FUNCTION_BLOCK "HOPPER"	// FB 1001
TITLE = HOPPER
//Creation:
//Date:            Author:                                               Version
//--------------------------------------------------------------------------------
//17.04.17          Ilia Bedniakov (ilia   )                             01.00.00
//
//Changes:
//No. Date:        Who       Description                           Mark   Version 
//--------------------------------------------------------------------------------
//01
//________________________________________________________________________________
//Function:
AUTHOR : ilia
VERSION : 0.1
VAR_INPUT
  in_HopperNumber : INT ;
  IF_FC_RotaryFeeder_DB : INT ;	//IF DB number
  IF_FC_RotaryFeeder_DW : INT ;	//start DW of IF structure
  SystemActive : BOOL ;	//system control on
  iLowLevelHopper : BOOL ;
  iRepRotaryFeeder : BOOL ;	//repair switch
  iRepVibrator1 : BOOL ;
  iRepVibrator2 : BOOL ;
  iFBVibrator1_on : BOOL ;
  iFBVibrator2_on : BOOL ;
  iFBRotaryFeeder_on : BOOL ;	//feedback
  iProductValve_open : BOOL ;	//feedback
  iSafetyRotaryFeeder_ok : BOOL ;	//safety switch
  iSafetyToolKeyControl : BOOL ;	//Tool control safety switch
  aFBRotaryFeeder : BOOL ;	//ack feedback fault
  aFBVibrator1 : BOOL ;
  aFBVibrator2 : BOOL ;
  aRepRotaryValve : BOOL ;	//ack repair switch
  aRepVibrator1 : BOOL ;
  aRepVibrator2 : BOOL ;
  aSafetyRotaryFeeder : BOOL ;	//ack safety switch
  aToolKeyControl : BOOL ;	//ack Tool Control
END_VAR
VAR_IN_OUT
  qRotaryFeeder_on : BOOL ;	//output
  qAPBRotaryFeeder : BOOL ;	//output
  qVibrator1 : BOOL ;
  qVibrator2 : BOOL ;
  fFBRotaryFeeder : BOOL ;	//feedback fault
  fFBVibrator1 : BOOL ;
  fFBVibrator2 : BOOL ;
  fRepRotaryFeeder : BOOL ;	//repair switch fault
  fRepVibrator1 : BOOL ;
  fRepVibrator2 : BOOL ;
  fSafetyRotaryFeeder : BOOL ;	//safety fault
  fToolKeyControl : BOOL ;	//rotary control fault
  fProductFlap : BOOL ;
END_VAR
VAR
  reserve_IO : ARRAY  [12 .. 49 ] OF BYTE ;
  HMI : STRUCT 	//Interface of HMI
   CMD : STRUCT
    reserve : BOOL ;
    Vibrator1_man_release : BOOL ;
    Vibrator2_man_release : BOOL ;
    reserve_3 : BOOL ;
    reserve_4 : BOOL ;
    reserve_5 : BOOL ;
    reserve_6 : BOOL ;
    reserve_7 : BOOL ;
    reserve_8 : BOOL ;
    reserve_9 : BOOL ;
    reserve_10 : BOOL ;
    reserve_11 : BOOL ;
    reserve_12 : BOOL ;
    reserve_13 : BOOL ;
    reserve_14 : BOOL ;
    reserve_15 : BOOL ;
   END_STRUCT ;
   STATE : STRUCT
    Active_Discharge : BOOL ;
    reserve_14 : BOOL ;
    reserve_12 : BOOL ;
    DischargingReleased : BOOL ;
    reserve : BOOL ;
    reserve_1 : BOOL ;
    reserve_2 : BOOL ;
    reserve_3 : BOOL ;
    reserve_4 : BOOL ;
    reserve_5 : BOOL ;
    reserve_6 : BOOL ;
    reserve_7 : BOOL ;
    reserve_8 : BOOL ;
    reserve_9 : BOOL ;
    reserve_10 : BOOL ;
    reserve_11 : BOOL ;
   END_STRUCT ;
   PARAM : STRUCT
    SetFrequency : REAL  := 3.000000e+001;
    DelayOn_RotaryValve : REAL  := 3.000000e+000;
    RestDischarge_Time : REAL  := 1.000000e+001;
    reserve_2 : REAL ;
    reserve_3 : INT ;
    reserve_4 : INT ;
    reserve_5 : INT ;
    reserve_6 : INT ;
    reserve_7 : INT ;
    reserve_8 : INT ;
    reserve_9 : REAL  := 1.200000e+002;
    reserve_10 : REAL  := 3.000000e+002;
    reserve_11 : REAL  := 5.000000e+000;
    reserve_12 : REAL  := 1.000000e+001;	//Minutes
    reserve_13 : REAL  := 1.000000e+001;
   END_STRUCT ;
   PV : STRUCT
    actFrequency : REAL ;
    DelayOn_RotaryValve : REAL ;
    RestDischarge_Time : REAL ;
    reserve : REAL ;
    reserve_1 : REAL ;
    reserve_2 : INT ;
    reserve_3 : INT ;
    reserve_4 : INT ;
    reserve_5 : INT ;
    reserve_6 : INT ;
    reserve_7 : INT ;
    reserve_8 : REAL ;
    reserve_9 : REAL ;
    reserve_10 : REAL ;
    reserve_11 : REAL ;	//Minutes
   END_STRUCT ;
  END_STRUCT ;
  PROD : STRUCT 	//Interface of Production
   FROM : STRUCT
    reserve : INT ;
    reserve_1 : INT ;
    reserve_2 : INT ;
    reserve_3 : INT ;
    reserve_4 : INT ;
    reserve_5 : REAL ;
    reserve_6 : REAL ;
    CMD : STRUCT
     reserve : BOOL ;
     reserve_1 : BOOL ;
     reserve_2 : BOOL ;
     reserve_3 : BOOL ;
     reserve_4 : BOOL ;
     reserve_5 : BOOL ;
     reserve_6 : BOOL ;
     reserve_7 : BOOL ;
     reserve_8 : BOOL ;
     reserve_9 : BOOL ;
     reserve_10 : BOOL ;
     reserve_11 : BOOL ;
     reserve_12 : BOOL ;
     reserve_13 : BOOL ;
     reserve_14 : BOOL ;
     reserve_15 : BOOL ;
    END_STRUCT ;
   END_STRUCT ;
   TO : STRUCT
    reserve : INT ;
    reserve_1 : INT ;
    reserve_2 : INT ;
    reserve_3 : INT ;
    reserve_4 : INT ;
    reserve_5 : REAL ;
    reserve_6 : REAL ;
    STATE : STRUCT
     reserve : BOOL ;
     reserve_1 : BOOL ;
     reserve_2 : BOOL ;
     reserve_3 : BOOL ;
     reserve_4 : BOOL ;
     reserve_5 : BOOL ;
     reserve_6 : BOOL ;
     reserve_7 : BOOL ;
     reserve_8 : BOOL ;
     reserve_9 : BOOL ;
     reserve_10 : BOOL ;
     reserve_11 : BOOL ;
     reserve_12 : BOOL ;
     reserve_13 : BOOL ;
     reserve_14 : BOOL ;
     reserve_15 : BOOL ;
    END_STRUCT ;
   END_STRUCT ;
   reserve : ARRAY  [40 .. 49 ] OF BYTE ;
  END_STRUCT ;
  IF_RECEIVER : STRUCT 	//Interface scale in storage location
   CONTROL : STRUCT
    Answer_DB : INT ;
    Answer_DW : INT ;
    reserve : REAL ;
    reserve_1 : INT ;
    reserve_2 : INT ;
    reserve_3 : INT ;
    reserve_4 : REAL ;
    CMD : STRUCT
     Request : BOOL ;
     Release : BOOL ;
     RECFull : BOOL ;
     reserve_11 : BOOL ;
     reserve_12 : BOOL ;
     reserve : BOOL ;
     reserve_1 : BOOL ;
     reserve_2 : BOOL ;
     reserve_3 : BOOL ;
     reserve_4 : BOOL ;
     reserve_5 : BOOL ;
     reserve_6 : BOOL ;
     reserve_7 : BOOL ;
     reserve_8 : BOOL ;
     reserve_9 : BOOL ;
     reserve_10 : BOOL ;
    END_STRUCT ;
   END_STRUCT ;
   STATUS : STRUCT
    reserve_1 : INT ;
    reserve_2 : INT ;
    reserve_3 : INT ;
    reserve_4 : INT ;
    reserve_5 : INT ;
    reserve_6 : REAL ;
    reserve_7 : REAL ;
    STATE : STRUCT
     Ready : BOOL ;
     Active : BOOL ;
     reserve : BOOL ;
     reserve_1 : BOOL ;
     reserve_2 : BOOL ;
     reserve_3 : BOOL ;
     reserve_4 : BOOL ;
     reserve_5 : BOOL ;
     reserve_6 : BOOL ;
     reserve_7 : BOOL ;
     reserve_8 : BOOL ;
     reserve_9 : BOOL ;
     reserve_10 : BOOL ;
     reserve_11 : BOOL ;
     reserve_12 : BOOL ;
     reserve_13 : BOOL ;
    END_STRUCT ;
   END_STRUCT ;
  END_STRUCT ;
  IF_FC_RotaryFeeder : STRUCT 	//Interface FC in active object
   STATUS : STRUCT
    ActualFrequency : REAL ;
    reserve : INT ;
    reserve_1 : INT ;
    reserve_2 : INT ;
    reserve_3 : INT ;
    reserve_4 : INT ;
    reserve_5 : REAL ;
    STATE : STRUCT
     Ready : BOOL ;
     Active : BOOL ;
     Fault : BOOL ;
     reserve : BOOL ;
     reserve_1 : BOOL ;
     reserve_2 : BOOL ;
     reserve_3 : BOOL ;
     reserve_4 : BOOL ;
     reserve_5 : BOOL ;
     reserve_6 : BOOL ;
     reserve_7 : BOOL ;
     reserve_8 : BOOL ;
     reserve_9 : BOOL ;
     reserve_10 : BOOL ;
     reserve_11 : BOOL ;
     reserve_12 : BOOL ;
    END_STRUCT ;
   END_STRUCT ;
   CONTROL : STRUCT
    Answer_DB : INT ;
    Answer_DW : INT ;
    Frequency_Set : REAL ;
    No_motor_data : INT ;
    reserve : INT ;
    reserve_1 : INT ;
    reserve_2 : REAL ;
    CMD : STRUCT
     Request : BOOL ;
     Release : BOOL ;
     Left_run : BOOL ;
     reserve : BOOL ;
     reserve_1 : BOOL ;
     reserve_2 : BOOL ;
     reserve_3 : BOOL ;
     reserve_4 : BOOL ;
     reserve_5 : BOOL ;
     reserve_6 : BOOL ;
     reserve_7 : BOOL ;
     reserve_8 : BOOL ;
     reserve_9 : BOOL ;
     reserve_10 : BOOL ;
     reserve_11 : BOOL ;
     reserve_12 : BOOL ;
    END_STRUCT ;
   END_STRUCT ;
  END_STRUCT ;
  reserve_IF : ARRAY  [280 .. 499 ] OF BYTE ;
  RotaryFeeder : STRUCT 	//motor object
   parameter : STRUCT
    motor_on : BOOL  := TRUE;	//activate motor structure
    clock_on : BOOL ;	//activate clock structure
    FC_on : BOOL  := TRUE;	//activate frequency converter structure
    hour_meter_on : BOOL ;	//activate hour meter
    reserve_4 : BOOL ;
    reserve_5 : BOOL ;
    reserve_6 : BOOL ;
    reserve_7 : BOOL ;
   END_STRUCT ;
   quit_motor : BOOL ;	//1 = quit motor on
   input_motor : BOOL ;	//1 = input motor on (return indication)
   motor_locked : BOOL ;	//1 = motor locked (in manual and auto mode) e.g. repair-/safety switch
   auto_mode_control : BOOL ;	//1 = release/control of motor in auto mode
   motor_in_operation : BOOL ;	//1 = signal motor in operation
   fault : BOOL ;	//1 = signal motor fault
   man_mode_to_SCADA : BOOL ;	//0 = Automatik Mode, 1 = Hand Mode
   man_mode_from_SCADA : BOOL ;	//0 = Automatik Mode, 1 = Hand Mode
   man_mode_control : BOOL ;	//1 = release/control of motor in manual mode (from SCADA)
   man_mode_locked : BOOL ;	//1 = change to manual mode locked, motor is in automatic use
   start_with_impulse : BOOL  := TRUE;	//1 = start cycle with impulse
   set_cycles_reached : BOOL ;	//1 = set number of cycles has been reached
   continous_clock : BOOL  := TRUE;	//1 = continous clock / 0 = set number of clocks
   simulation : BOOL ;	//1 = simulation of object
   release_clock : BOOL ;	//1 = release bit for clock FC
   quit_clock : BOOL ;	//quit for clock FC, if release_clock = TRUE
   set_time_fault : INT  := 5;	//fault evaluation time in seconds
   actual_time_fault : INT ;	//actual fault evaluation time in seconds
   impulse_time : REAL  := 5.000000e+000;	//impulse time for clock in seconds
   break_time : REAL  := 5.000000e+000;	//break time for clock in seconds
   time_counter : REAL ;	//time counter (elapsed time)
   set_cycles : INT ;	//number of clocks if not continous clock
   clock_counter : INT ;	//clock counter
   FCs : STRUCT 	//frequency converter
    FC_in_operation : BOOL ;	//1 = FU in Betrieb
    fault : BOOL ;	//1 = FC fault
    set_revolutions_man_mode : INT ;	//revolutions in permille in manual mode
    actual_revolutions : INT ;	//actual revolutions FC in man/auto mode
   END_STRUCT ;
   hour_meter : STRUCT 	//hour meter
    reset : BOOL ;	//reset hour meter
    warning : BOOL ;	//warning time exceeded
    alarm : BOOL ;	//alarm time exceeded
    actual_operating_hours : REAL ;	//actual operating hours (in hours)
    set_time_warning : REAL ;	//set time for warning (in hours)
    set_time_alarm : REAL ;	//set time for alarm (in hours)
    second_counter_oh : INT ;	//seconds of the actual operatin hours
   END_STRUCT ;
   system_on : BOOL ;	//system released resepectively system area released after emergency stopping
   object_state : INT ;	//1=grey; 5=green; 9=white; 15=yellow; 16=red
  END_STRUCT ;
  APBRotaryFeeder : STRUCT 	//valve object with 1Q and 0-2I
   parameter : STRUCT
    valve_on : BOOL  := TRUE;	//activate valve structure
    clock_on : BOOL ;	//activate clock structure
    reserve_3 : BOOL ;
    switching_number_on : BOOL ;	//activate switching number counter
    reserve_4 : BOOL ;
    parameter_1Q : BOOL  := TRUE;	//valve type with 1 quit 0 inputs
    parameter_1Q_1I : BOOL ;	//valve type with 1 quit 1 input (=)
    parameter_1Q_1IN : BOOL ;	//valve type with 1 quit 1 input (<>)
    parameter_1Q_2I : BOOL ;	//valve type with 1 quit 2 inputs
    parameter_text_pos_1 : BOOL ;
    parameter_text_straight : BOOL ;
    parameter_text_inverse : BOOL ;	//select text inverse = "close/open" or "bypass/convey" aso.
    parameter_text_open : BOOL ;	//select text quit = "open/close"
    parameter_text_convey : BOOL ;	//select text quit = "convey/bypass"
    parameter_text_on : BOOL  := TRUE;	//select text quit = "on/off"
    parameter_text_up : BOOL ;	//select text quit = "up/down"
   END_STRUCT ;
   quit_valve : BOOL ;	//1 = quit valve
   input_valve_set : BOOL ;	//1 = input valve, if quit valve set
   input_valve_not_set : BOOL ;	//1 = input valve, if quit valve not set
   auto_mode_control : BOOL ;	//1 = release/control of valve in auto mode
   valve_in_operation : BOOL ;	//1 = signal valve in operation
   fault : BOOL ;	//1 = signal valve fault
   man_mode_to_SCADA : BOOL ;	//0 = automatic mode , 1 = manual mode
   man_mode_from_SCADA : BOOL ;	//0 = automatic mode , 1 = manual mode
   man_mode_control : BOOL ;	//1 = release/control of valve in manual mode (from SCADA)
   man_mode_locked : BOOL ;	//1 = change to manual mode locked, valve is in automatic use
   start_with_impulse : BOOL ;	//1 = start cycle with impluse
   set_cycles_reached : BOOL ;	//1 = set number of cycles has been reached
   continous_clock : BOOL ;	//1 = continous clock / 0 = set number of clocks
   simulation : BOOL ;	//1 = simulation of object
   release_clock : BOOL ;	//1 = release bit for clock FC
   quit_clock : BOOL ;	//quit for clock FC, if release_clock = TRUE
   set_time_fault : INT  := 5;	//fault evaluation time in seconds
   actual_time_fault : INT ;	//actual fault evaluation time in seconds
   impulse_time : REAL  := 5.000000e+000;	//impulse time for clock in seconds
   break_time : REAL  := 5.000000e+000;	//break time for clock in seconds
   time_counter : REAL ;	//time counter (elapsed time)
   set_cycles : INT ;	//number of clocks if not continous clock
   clock_counter : INT ;	//clock counter
   switching_number_counter : STRUCT 	//switching number counter
    reset : BOOL ;	//reset switching number counter
    warning : BOOL ;	//warning number exceeded
    alarm : BOOL ;	//alarm number exceeded
    flank_flag : BOOL ;	//internal flag
    actual_switching_number : REAL ;	//actual switching number
    set_number_warning : REAL ;	//set number for warning
    set_number_alarm : REAL ;	//set number for alarm
   END_STRUCT ;
   set_time_in_operation : INT ;	//1IoO: set time for delay of "valve in operation"
   real_time_in_operation : INT ;	//1IoO: real time for delay of "valve in operation"
   system_on : BOOL ;	//system released resepectively system area released after emergency stopping
   reserve : ARRAY  [44 .. 47 ] OF BYTE ;
   object_state : INT ;	//1=grey; 5=green; 9=white; 15=yellow; 16=red
  END_STRUCT ;
  Vibrator1 : STRUCT 	//motor object
   parameter : STRUCT
    motor_on : BOOL  := TRUE;	//activate motor structure
    clock_on : BOOL  := TRUE;	//activate clock structure
    FC_on : BOOL ;	//activate frequency converter structure
    hour_meter_on : BOOL ;	//activate hour meter
    reserve_4 : BOOL ;
    reserve_5 : BOOL ;
    reserve_6 : BOOL ;
    reserve_7 : BOOL ;
   END_STRUCT ;
   quit_motor : BOOL ;	//1 = quit motor on
   input_motor : BOOL ;	//1 = input motor on (return indication)
   motor_locked : BOOL ;	//1 = motor locked (in manual and auto mode) e.g. repair-/safety switch
   auto_mode_control : BOOL ;	//1 = release/control of motor in auto mode
   motor_in_operation : BOOL ;	//1 = signal motor in operation
   fault : BOOL ;	//1 = signal motor fault
   man_mode_to_SCADA : BOOL ;	//0 = Automatik Mode, 1 = Hand Mode
   man_mode_from_SCADA : BOOL ;	//0 = Automatik Mode, 1 = Hand Mode
   man_mode_control : BOOL ;	//1 = release/control of motor in manual mode (from SCADA)
   man_mode_locked : BOOL ;	//1 = change to manual mode locked, motor is in automatic use
   start_with_impulse : BOOL  := TRUE;	//1 = start cycle with impulse
   set_cycles_reached : BOOL ;	//1 = set number of cycles has been reached
   continous_clock : BOOL  := TRUE;	//1 = continous clock / 0 = set number of clocks
   simulation : BOOL ;	//1 = simulation of object
   release_clock : BOOL  := TRUE;	//1 = release bit for clock FC
   quit_clock : BOOL ;	//quit for clock FC, if release_clock = TRUE
   set_time_fault : INT  := 5;	//fault evaluation time in seconds
   actual_time_fault : INT ;	//actual fault evaluation time in seconds
   impulse_time : REAL  := 5.000000e+000;	//impulse time for clock in seconds
   break_time : REAL  := 5.000000e+000;	//break time for clock in seconds
   time_counter : REAL ;	//time counter (elapsed time)
   set_cycles : INT ;	//number of clocks if not continous clock
   clock_counter : INT ;	//clock counter
   FCs : STRUCT 	//frequency converter
    FC_in_operation : BOOL ;	//1 = FU in Betrieb
    fault : BOOL ;	//1 = FC fault
    set_revolutions_man_mode : INT ;	//revolutions in permille in manual mode
    actual_revolutions : INT ;	//actual revolutions FC in man/auto mode
   END_STRUCT ;
   hour_meter : STRUCT 	//hour meter
    reset : BOOL ;	//reset hour meter
    warning : BOOL ;	//warning time exceeded
    alarm : BOOL ;	//alarm time exceeded
    actual_operating_hours : REAL ;	//actual operating hours (in hours)
    set_time_warning : REAL ;	//set time for warning (in hours)
    set_time_alarm : REAL ;	//set time for alarm (in hours)
    second_counter_oh : INT ;	//seconds of the actual operatin hours
   END_STRUCT ;
   system_on : BOOL ;	//system released resepectively system area released after emergency stopping
   object_state : INT ;	//1=grey; 5=green; 9=white; 15=yellow; 16=red
  END_STRUCT ;
  Vibrator2 : STRUCT 	//motor object
   parameter : STRUCT
    motor_on : BOOL  := TRUE;	//activate motor structure
    clock_on : BOOL  := TRUE;	//activate clock structure
    FC_on : BOOL ;	//activate frequency converter structure
    hour_meter_on : BOOL ;	//activate hour meter
    reserve_4 : BOOL ;
    reserve_5 : BOOL ;
    reserve_6 : BOOL ;
    reserve_7 : BOOL ;
   END_STRUCT ;
   quit_motor : BOOL ;	//1 = quit motor on
   input_motor : BOOL ;	//1 = input motor on (return indication)
   motor_locked : BOOL ;	//1 = motor locked (in manual and auto mode) e.g. repair-/safety switch
   auto_mode_control : BOOL ;	//1 = release/control of motor in auto mode
   motor_in_operation : BOOL ;	//1 = signal motor in operation
   fault : BOOL ;	//1 = signal motor fault
   man_mode_to_SCADA : BOOL ;	//0 = Automatik Mode, 1 = Hand Mode
   man_mode_from_SCADA : BOOL ;	//0 = Automatik Mode, 1 = Hand Mode
   man_mode_control : BOOL ;	//1 = release/control of motor in manual mode (from SCADA)
   man_mode_locked : BOOL ;	//1 = change to manual mode locked, motor is in automatic use
   start_with_impulse : BOOL  := TRUE;	//1 = start cycle with impulse
   set_cycles_reached : BOOL ;	//1 = set number of cycles has been reached
   continous_clock : BOOL  := TRUE;	//1 = continous clock / 0 = set number of clocks
   simulation : BOOL ;	//1 = simulation of object
   release_clock : BOOL  := TRUE;	//1 = release bit for clock FC
   quit_clock : BOOL ;	//quit for clock FC, if release_clock = TRUE
   set_time_fault : INT  := 5;	//fault evaluation time in seconds
   actual_time_fault : INT ;	//actual fault evaluation time in seconds
   impulse_time : REAL  := 5.000000e+000;	//impulse time for clock in seconds
   break_time : REAL  := 5.000000e+000;	//break time for clock in seconds
   time_counter : REAL ;	//time counter (elapsed time)
   set_cycles : INT ;	//number of clocks if not continous clock
   clock_counter : INT ;	//clock counter
   FCs : STRUCT 	//frequency converter
    FC_in_operation : BOOL ;	//1 = FU in Betrieb
    fault : BOOL ;	//1 = FC fault
    set_revolutions_man_mode : INT ;	//revolutions in permille in manual mode
    actual_revolutions : INT ;	//actual revolutions FC in man/auto mode
   END_STRUCT ;
   hour_meter : STRUCT 	//hour meter
    reset : BOOL ;	//reset hour meter
    warning : BOOL ;	//warning time exceeded
    alarm : BOOL ;	//alarm time exceeded
    actual_operating_hours : REAL ;	//actual operating hours (in hours)
    set_time_warning : REAL ;	//set time for warning (in hours)
    set_time_alarm : REAL ;	//set time for alarm (in hours)
    second_counter_oh : INT ;	//seconds of the actual operatin hours
   END_STRUCT ;
   system_on : BOOL ;	//system released resepectively system area released after emergency stopping
   object_state : INT ;	//1=grey; 5=green; 9=white; 15=yellow; 16=red
  END_STRUCT ;
  LevelIndicators : STRUCT
   LowLevelHopper : STRUCT
    input : BOOL ;
    debounced_covered : BOOL ;
    helpmarker : BOOL ;
    fault : BOOL ;
   END_STRUCT ;
  END_STRUCT ;
  reserve_Cmod : ARRAY  [702 .. 799 ] OF BYTE ;
  TIMES : STRUCT 	//ten timers
   TON_FC_RotaryValve : STRUCT
    IN : BOOL ;
    RST : BOOL ;
    IMP : BOOL ;
    Q : BOOL ;
    PT : REAL ;
    ET : REAL ;
   END_STRUCT ;
   TOF_FC_RotaryValve : STRUCT
    IN : BOOL ;
    RST : BOOL ;
    IMP : BOOL ;
    Q : BOOL ;
    PT : REAL ;
    ET : REAL ;
   END_STRUCT ;
   TOF_RotaryValve : STRUCT
    IN : BOOL ;
    RST : BOOL ;
    IMP : BOOL ;
    Q : BOOL ;
    PT : REAL ;
    ET : REAL ;
   END_STRUCT ;
   TOF_APBRotaryValve : STRUCT
    IN : BOOL ;
    RST : BOOL ;
    IMP : BOOL ;
    Q : BOOL ;
    PT : REAL ;
    ET : REAL ;
   END_STRUCT ;
   TON_WRestDischarge : STRUCT 	//with rest discharge
    IN : BOOL ;
    RST : BOOL ;
    IMP : BOOL ;
    Q : BOOL ;
    PT : REAL ;
    ET : REAL ;
   END_STRUCT ;
   TON_DelayStart : STRUCT 	//with rest discharge
    IN : BOOL ;
    RST : BOOL ;
    IMP : BOOL ;
    Q : BOOL ;
    PT : REAL ;
    ET : REAL ;
   END_STRUCT ;
  END_STRUCT ;
  SEQUENCES : STRUCT
   Filling : STRUCT
    AUTO : BOOL ;
    MANUAL : BOOL ;
    LOCKED : BOOL ;
    reserve : BOOL ;
    reserve_1 : BOOL ;
    reserve_2 : BOOL ;
    reserve_3 : BOOL ;
    reserve_4 : BOOL ;
    reserve_5 : BOOL ;
    reserve_6 : BOOL ;
    reserve_7 : BOOL ;
    reserve_8 : BOOL ;
    reserve_9 : BOOL ;
    reserve_10 : BOOL ;
    reserve_11 : BOOL ;
    reserve_12 : BOOL ;
   END_STRUCT ;
   Discharging : STRUCT
    AUTO : BOOL ;
    MANUAL : BOOL ;
    LOCKED : BOOL ;
    RELEASE : BOOL ;
    reserve_1 : BOOL ;
    reserve_2 : BOOL ;
    reserve_3 : BOOL ;
    reserve_4 : BOOL ;
    reserve_5 : BOOL ;
    reserve_6 : BOOL ;
    reserve_7 : BOOL ;
    reserve_8 : BOOL ;
    reserve_9 : BOOL ;
    reserve_10 : BOOL ;
    reserve_11 : BOOL ;
    reserve_12 : BOOL ;
   END_STRUCT ;
   reserve : ARRAY  [4 .. 99 ] OF BYTE ;
  END_STRUCT ;
  INTERNAL : STRUCT
   IF : STRUCT
    FC_RotaryValve_ready : BOOL ;
    reserve : BOOL ;
    reserve_1 : BOOL ;
    reserve_2 : BOOL ;
    reserve_3 : BOOL ;
    reserve_4 : BOOL ;
    reserve_5 : BOOL ;
    reserve_6 : BOOL ;
    reserve_7 : BOOL ;
    reserve_8 : BOOL ;
    reserve_9 : BOOL ;
    reserve_10 : BOOL ;
    reserve_11 : BOOL ;
    reserve_12 : BOOL ;
    reserve_13 : BOOL ;
    reserve_14 : BOOL ;
   END_STRUCT ;
   Flags : STRUCT
    second_vibro_exist : BOOL ;
    reserve_1 : BOOL ;
    reserve_2 : BOOL ;
    reserve_3 : BOOL ;
    reserve_4 : BOOL ;
    reserve_5 : BOOL ;
    reserve_6 : BOOL ;
    reserve_7 : BOOL ;
    reserve_8 : BOOL ;
    reserve_9 : BOOL ;
    reserve_10 : BOOL ;
    reserve_10_5 : BOOL ;
    reserve_10_4 : BOOL ;
    reserve_10_3 : BOOL ;
    reserve_10_2 : BOOL ;
    reserve_10_1 : BOOL ;
   END_STRUCT ;
   Instance_DB_number : INT ;
  END_STRUCT ;
END_VAR
BEGIN
NETWORK
TITLE = ---- instance DB ----
      L     0;
      L     DINO;
      ==I;
      BEC;
      T     #INTERNAL.Instance_DB_number;
NETWORK
TITLE = ---- Sequence status ----
NETWORK
TITLE = Sequence discharging auto
      A     #IF_RECEIVER.CONTROL.CMD.Request;
      AN    #fToolKeyControl;
      AN    #fSafetyRotaryFeeder;
      AN    #SEQUENCES.Discharging.LOCKED;
      =     #SEQUENCES.Discharging.AUTO;
NETWORK
TITLE = Sequence discharging manual
      O     #RotaryFeeder.man_mode_to_SCADA;
      AN    #SEQUENCES.Discharging.AUTO;
      =     #SEQUENCES.Discharging.MANUAL;
NETWORK
TITLE = Sequence discharging locked
      O     #SEQUENCES.Discharging.MANUAL;
      ON    #SystemActive;
      =     #SEQUENCES.Discharging.LOCKED;
NETWORK
TITLE = ---- General status ----
NETWORK
TITLE = rotary valve safety switch & maintenance switch
//safety switch
      A     #iSafetyRotaryFeeder_ok;
      A     #aSafetyRotaryFeeder;
      R     #fSafetyRotaryFeeder;
      AN    #iSafetyRotaryFeeder_ok;
      S     #fSafetyRotaryFeeder;
//maintenance switch
      A     #iRepRotaryFeeder;
      A     #aRepRotaryValve;
      R     #fRepRotaryFeeder;
      O     #RotaryFeeder.auto_mode_control;
      O     #RotaryFeeder.man_mode_control;
      AN    #iRepRotaryFeeder;
      S     #fRepRotaryFeeder;
NETWORK
TITLE = Discharging: Second vibrator exist??
      A(;
      L     #in_HopperNumber;
      L     2;
      ==I;
      );
      =     #INTERNAL.Flags.second_vibro_exist;
NETWORK
TITLE = vibrator 1 maintenance switch
//maintenance switch
      A     #iRepVibrator1;
      A     #aRepVibrator1;
      R     #fRepVibrator1;
      O     #Vibrator1.auto_mode_control;
      O     #Vibrator1.man_mode_control;
      AN    #iRepVibrator1;
      S     #fRepVibrator1;
NETWORK
TITLE = vibrator 2 maintenance switch
//maintenance switch
      A     #iRepVibrator2;
      A     #aRepVibrator2;
      ON    #INTERNAL.Flags.second_vibro_exist;
      R     #fRepVibrator2;
      O     #Vibrator2.auto_mode_control;
      O     #Vibrator2.man_mode_control;
      AN    #iRepVibrator2;
      A     #INTERNAL.Flags.second_vibro_exist;
      S     #fRepVibrator2;
NETWORK
TITLE = rotor control RV 
      A     #iSafetyToolKeyControl;
      A     #aToolKeyControl;
      R     #fToolKeyControl;
      O     #RotaryFeeder.auto_mode_control;
      O     #RotaryFeeder.man_mode_control;
      AN    #iSafetyToolKeyControl;
      S     #fToolKeyControl;
NETWORK
TITLE = Low/Full Level Sensor
      AN    #iLowLevelHopper;
      =     #LevelIndicators.LowLevelHopper.input;
      CALL  "FC14 Debounce Indicator" (
           Eingang                  := #LevelIndicators.LowLevelHopper.input,
           Takt                     := "M 1.6 ClckDdebounceIndic",
           Folgemerker              := #LevelIndicators.LowLevelHopper.helpmarker,
           Eingang_entprellt        := #LevelIndicators.LowLevelHopper.debounced_covered);
NETWORK
TITLE = ---- Sequence Discharging ----
NETWORK
TITLE = Discharging: discharge released
      A     #SystemActive;
      A     #IF_RECEIVER.CONTROL.CMD.Request;
      =     #SEQUENCES.Discharging.RELEASE;
      A     #SEQUENCES.Discharging.RELEASE;
      =     #HMI.STATE.DischargingReleased;
NETWORK
TITLE = fault: manual flap not open
      A     #IF_RECEIVER.CONTROL.CMD.Request;
      AN    #iProductValve_open;
      =     #fProductFlap;
NETWORK
TITLE = Discharging: request to FC dosing screw
      A(;
      A     #SEQUENCES.Discharging.AUTO;
      A     #IF_RECEIVER.CONTROL.CMD.Request;
      AN    #RotaryFeeder.man_mode_to_SCADA;
      O;
      A     #RotaryFeeder.man_mode_to_SCADA;
      A     #RotaryFeeder.man_mode_control;
      );
      AN    #fSafetyRotaryFeeder;
      AN    #fToolKeyControl;
      AN    #fRepRotaryFeeder;
      O;
      A     #RotaryFeeder.FCs.FC_in_operation;
      =     #IF_FC_RotaryFeeder.CONTROL.CMD.Request;
NETWORK
TITLE = Discharging: ready to receiver
      A     #SEQUENCES.Discharging.AUTO;
      A     #IF_RECEIVER.CONTROL.CMD.Request;
      A     #IF_FC_RotaryFeeder.STATUS.STATE.Ready;
      =     #TIMES.TON_DelayStart.IN;
      CALL  "FC3 Cycle generator" (
           in_Freigabe              := #TIMES.TON_DelayStart.IN,
           in_Reset                 := #TIMES.TON_DelayStart.RST,
           in_Impuls                := "M 1.7 Cycle Timer-FC",
           in_Impulszeit_in_100ms   := "MW 6 Timer Val Cycle FCs",
           in_Verzoegerungsart      := B#16#45,
           in_Verzoegerungszeit     := #HMI.PARAM.DelayOn_RotaryValve,
           io_Ausgangssignal        := #TIMES.TON_DelayStart.Q,
           io_Zeitzaehler           := #HMI.PV.DelayOn_RotaryValve);
      A     #TIMES.TON_DelayStart.Q;
      =     #IF_RECEIVER.STATUS.STATE.Ready;
NETWORK
TITLE = Discharging: release air purged bearing
      A     #SEQUENCES.Discharging.AUTO;
      A     #IF_RECEIVER.CONTROL.CMD.Request;
      A     #IF_FC_RotaryFeeder.STATUS.STATE.Ready;
      A     #IF_RECEIVER.STATUS.STATE.Ready;
      A     #IF_RECEIVER.CONTROL.CMD.Release;
      AN    #fToolKeyControl;
      AN    #fSafetyRotaryFeeder;
      =     #TIMES.TOF_APBRotaryValve.IN;
      ON    #SystemActive;
      =     #TIMES.TOF_APBRotaryValve.RST;
      CALL  "FC3 Cycle generator" (
           in_Freigabe              := #TIMES.TOF_APBRotaryValve.IN,
           in_Reset                 := #TIMES.TOF_APBRotaryValve.RST,
           in_Impuls                := "M 1.7 Cycle Timer-FC",
           in_Impulszeit_in_100ms   := "MW 6 Timer Val Cycle FCs",
           in_Verzoegerungsart      := B#16#41,
           in_Verzoegerungszeit     := 2.000000e+00,
           io_Ausgangssignal        := #TIMES.TOF_APBRotaryValve.Q,
           io_Zeitzaehler           := #TIMES.TOF_APBRotaryValve.ET);	// 3.000000e+000
      A     #TIMES.TOF_APBRotaryValve.Q;
      =     #APBRotaryFeeder.auto_mode_control;
NETWORK
TITLE = Discharging: air purging bearing object
      A     #SEQUENCES.Discharging.AUTO;
      AN    "Service mode lock auto";
      =     #APBRotaryFeeder.man_mode_locked;
      CALL  "FC21 Valve 10-2I" (
           in_Ventil_Typ            := 0,
           in_Handbedienung_erlaubt := TRUE,
           in_Quitt_Stoerung_noetig := FALSE,
           in_Quitt_Stoerung        := FALSE,
           in_Anlage_ein            := #SystemActive,
           in_Ansteuerung_Ventil    := #APBRotaryFeeder.auto_mode_control,
           in_Eingang_angesteuert   := #APBRotaryFeeder.input_valve_set,
           in_Eingang_nicht_angest  := #APBRotaryFeeder.input_valve_not_set,
           io_Ausgang_Ventil        := #qAPBRotaryFeeder,
           io_Ventil_in_Betrieb     := #APBRotaryFeeder.valve_in_operation,
           io_Stoerung              := #APBRotaryFeeder.fault,
           io_Ventilstruktur        := #APBRotaryFeeder);
NETWORK
TITLE = Discharging: release rotary valve
      A     #SEQUENCES.Discharging.AUTO;
      A     #IF_RECEIVER.CONTROL.CMD.Request;
      A     #IF_FC_RotaryFeeder.STATUS.STATE.Ready;
      A     #IF_RECEIVER.STATUS.STATE.Ready;
      A     #IF_RECEIVER.CONTROL.CMD.Release;
      A     #APBRotaryFeeder.valve_in_operation;
      =     #TIMES.TOF_RotaryValve.IN;
      ON    #iRepRotaryFeeder;
      ON    #SystemActive;
      =     #TIMES.TOF_RotaryValve.RST;
      CALL  "FC3 Cycle generator" (
           in_Freigabe              := #TIMES.TOF_RotaryValve.IN,
           in_Reset                 := #TIMES.TOF_RotaryValve.RST,
           in_Impuls                := "M 1.7 Cycle Timer-FC",
           in_Impulszeit_in_100ms   := "MW 6 Timer Val Cycle FCs",
           in_Verzoegerungsart      := B#16#41,
           in_Verzoegerungszeit     := 3.000000e+00,
           io_Ausgangssignal        := #TIMES.TOF_RotaryValve.Q,
           io_Zeitzaehler           := #TIMES.TOF_RotaryValve.ET);
      A     #TIMES.TOF_RotaryValve.Q;
      =     #RotaryFeeder.auto_mode_control;
NETWORK
TITLE = Discharging: Rotary Valve Object
      O     #SEQUENCES.Discharging.AUTO;
      AN    "Service mode lock auto";
      =     #RotaryFeeder.man_mode_locked;
      O     #fSafetyRotaryFeeder;
      O     #fToolKeyControl;
      O     #fRepRotaryFeeder;
      O     #IF_RECEIVER.CONTROL.CMD.RECFull;
      =     #RotaryFeeder.motor_locked;
//if FC not ready, reset man mode to SCADA and man mode control
      AN    #INTERNAL.IF.FC_RotaryValve_ready;
      R     #RotaryFeeder.man_mode_to_SCADA;
      R     #RotaryFeeder.man_mode_control;
      CALL  "FC20 Motor 1O1I" (
           in_Handbedienung_erlaubt := TRUE,
           in_Quitt_Stoerung_noetig := TRUE,
           in_Anlage_ein            := #SystemActive,
           in_Quitt_Stoerung        := #aFBRotaryFeeder,
           in_Ansteuerung_Motor     := #RotaryFeeder.auto_mode_control,
           in_Eingang_Motor         := #iFBRotaryFeeder_on,
           io_Ausgang_Motor         := #qRotaryFeeder_on,
           io_Motor_in_Betrieb      := #RotaryFeeder.motor_in_operation,
           io_Stoerung              := #fFBRotaryFeeder,
           io_Motorstruktur         := #RotaryFeeder);
NETWORK
TITLE = Discharging: TON Timer for FC Rotary Valve 
//on delay FC 
      A     #RotaryFeeder.motor_in_operation;
      =     #TIMES.TON_FC_RotaryValve.IN;
      ON    #SystemActive;
      =     #TIMES.TON_FC_RotaryValve.RST;
      CALL  "FC3 Cycle generator" (
           in_Freigabe              := #TIMES.TON_FC_RotaryValve.IN,
           in_Reset                 := #TIMES.TON_FC_RotaryValve.RST,
           in_Impuls                := "M 1.7 Cycle Timer-FC",
           in_Impulszeit_in_100ms   := "MW 6 Timer Val Cycle FCs",
           in_Verzoegerungsart      := B#16#45,
           in_Verzoegerungszeit     := 2.000000e+00,
           io_Ausgangssignal        := #TIMES.TON_FC_RotaryValve.Q,
           io_Zeitzaehler           := #TIMES.TON_FC_RotaryValve.ET);
NETWORK
TITLE = Discharging: TOF Timer for FC Rotary Valve 
//on delay FC 
      A     #RotaryFeeder.motor_in_operation;
      =     #TIMES.TON_FC_RotaryValve.IN;
      ON    #SystemActive;
      =     #TIMES.TON_FC_RotaryValve.RST;
      CALL  "FC3 Cycle generator" (
           in_Freigabe              := #TIMES.TOF_FC_RotaryValve.IN,
           in_Reset                 := #TIMES.TOF_FC_RotaryValve.RST,
           in_Impuls                := "M 1.7 Cycle Timer-FC",
           in_Impulszeit_in_100ms   := "MW 6 Timer Val Cycle FCs",
           in_Verzoegerungsart      := B#16#41,
           in_Verzoegerungszeit     := 1.000000e+00,
           io_Ausgangssignal        := #TIMES.TOF_FC_RotaryValve.Q,
           io_Zeitzaehler           := #TIMES.TOF_FC_RotaryValve.ET);
NETWORK
TITLE = Discharging: release FC dosing screw
      A(;
      A     #SEQUENCES.Discharging.AUTO;
      A     #IF_RECEIVER.CONTROL.CMD.Release;
      A     #APBRotaryFeeder.valve_in_operation;
      AN    #RotaryFeeder.man_mode_to_SCADA;
      O;
      A     #RotaryFeeder.man_mode_to_SCADA;
      A     #RotaryFeeder.man_mode_control;
      );
      A     #IF_FC_RotaryFeeder.STATUS.STATE.Ready;
      A(;
      A     #TIMES.TON_FC_RotaryValve.Q;
      O;
      AN    #RotaryFeeder.motor_in_operation;
      A     #TIMES.TOF_FC_RotaryValve.Q;
      );
      AN    #fSafetyRotaryFeeder;
      AN    #fToolKeyControl;
      AN    #fRepRotaryFeeder;
      =     #IF_FC_RotaryFeeder.CONTROL.CMD.Release;
NETWORK
TITLE = Discharging: data exchange with FC dosing screw
//dosing speed
      L     #HMI.PARAM.SetFrequency;	//auto
      A     #RotaryFeeder.man_mode_to_SCADA;
      JCN   RVA;	// rotary valve auto
      L     #RotaryFeeder.FCs.set_revolutions_man_mode;	//manual
      ITD;
      DTR;
      L     1.000000e+01;
      /R;
RVA:  T     #IF_FC_RotaryFeeder.CONTROL.Frequency_Set;
//FC in operation
      A     #IF_FC_RotaryFeeder.STATUS.STATE.Active;
      =     #RotaryFeeder.FCs.FC_in_operation;
//FC fault
      A     #IF_FC_RotaryFeeder.STATUS.STATE.Fault;
      =     #RotaryFeeder.FCs.fault;
//actual frequency
      L     #IF_FC_RotaryFeeder.STATUS.ActualFrequency;
      L     1.000000e+01;
      *R;
      RND;
      T     #RotaryFeeder.FCs.actual_revolutions;
      L     #IF_FC_RotaryFeeder.STATUS.ActualFrequency;
      T     #HMI.PV.actFrequency;
NETWORK
TITLE = Discharging: rest discharging
      AN    #LevelIndicators.LowLevelHopper.debounced_covered;
      A     #SEQUENCES.Discharging.RELEASE;
      =     #TIMES.TON_WRestDischarge.IN;
      CALL  "FC3 Cycle generator" (
           in_Freigabe              := #TIMES.TON_WRestDischarge.IN,
           in_Reset                 := #TIMES.TON_WRestDischarge.RST,
           in_Impuls                := "M 1.7 Cycle Timer-FC",
           in_Impulszeit_in_100ms   := "MW 6 Timer Val Cycle FCs",
           in_Verzoegerungsart      := B#16#45,
           in_Verzoegerungszeit     := #HMI.PARAM.RestDischarge_Time,
           io_Ausgangssignal        := #TIMES.TON_WRestDischarge.Q,
           io_Zeitzaehler           := #TIMES.TON_WRestDischarge.ET);
      L     #TIMES.TON_WRestDischarge.ET;
      T     #HMI.PV.RestDischarge_Time;
NETWORK
TITLE = Discharging: release auto vibrator 1 (bottom)
      A     #SEQUENCES.Discharging.AUTO;
      A     #IF_RECEIVER.CONTROL.CMD.Release;
      A     #RotaryFeeder.motor_in_operation;
      A(;
      AN    #INTERNAL.Flags.second_vibro_exist;	// HP01
      A     #TIMES.TON_WRestDischarge.Q;
      O;
      A     #INTERNAL.Flags.second_vibro_exist;	//HP02
      A     #iProductValve_open;
//      A     #TIMES.TON_WRestDischarge.Q
      );
      O;
      A     #SEQUENCES.Discharging.AUTO;
      A     #HMI.CMD.Vibrator1_man_release;
      =     #Vibrator1.auto_mode_control;
NETWORK
TITLE = Discharging: vibromotor motor 1 object
      O     #SEQUENCES.Discharging.AUTO;
      AN    "Service mode lock auto";
      =     #Vibrator1.man_mode_locked;
      A     #fRepVibrator1;
      =     #Vibrator1.motor_locked;
      CALL  "FC20 Motor 1O1I" (
           in_Handbedienung_erlaubt := TRUE,
           in_Quitt_Stoerung_noetig := TRUE,
           in_Anlage_ein            := #SystemActive,
           in_Quitt_Stoerung        := #aFBVibrator1,
           in_Ansteuerung_Motor     := #Vibrator1.auto_mode_control,
           in_Eingang_Motor         := #iFBVibrator1_on,
           io_Ausgang_Motor         := #qVibrator1,
           io_Motor_in_Betrieb      := #Vibrator1.motor_in_operation,
           io_Stoerung              := #fFBVibrator1,
           io_Motorstruktur         := #Vibrator1);
NETWORK
TITLE = Discharging: release auto vibrator 2
      A     #SEQUENCES.Discharging.AUTO;
      A     #INTERNAL.Flags.second_vibro_exist;
      A(;
      A     #IF_RECEIVER.CONTROL.CMD.Release;
      A     #RotaryFeeder.motor_in_operation;
      A     #TIMES.TON_WRestDischarge.Q;
      O;
      A     #HMI.CMD.Vibrator2_man_release;
      );
      =     #Vibrator2.auto_mode_control;
      AN    #SEQUENCES.Discharging.AUTO;
      R     #HMI.CMD.Vibrator1_man_release;
      R     #HMI.CMD.Vibrator2_man_release;
NETWORK
TITLE = Discharging: vibromotor motor 2 object
      A     #SEQUENCES.Discharging.AUTO;
      AN    "Service mode lock auto";
      =     #Vibrator2.man_mode_locked;
      A     #fRepVibrator2;
      =     #Vibrator2.motor_locked;
      CALL  "FC20 Motor 1O1I" (
           in_Handbedienung_erlaubt := TRUE,
           in_Quitt_Stoerung_noetig := TRUE,
           in_Anlage_ein            := #SystemActive,
           in_Quitt_Stoerung        := #aFBVibrator2,
           in_Ansteuerung_Motor     := #Vibrator2.auto_mode_control,
           in_Eingang_Motor         := #iFBVibrator2_on,
           io_Ausgang_Motor         := #qVibrator2,
           io_Motor_in_Betrieb      := #Vibrator2.motor_in_operation,
           io_Stoerung              := #fFBVibrator2,
           io_Motorstruktur         := #Vibrator2);
      NOP   0;
NETWORK
TITLE = Active to VISU
      A     #RotaryFeeder.auto_mode_control;
      A     #IF_FC_RotaryFeeder.STATUS.STATE.Active;
      =     #IF_RECEIVER.STATUS.STATE.Active;
      A     #IF_RECEIVER.STATUS.STATE.Active;
      =     #HMI.STATE.Active_Discharge;
NETWORK
TITLE = ---- interface ----
NETWORK
TITLE = Receiver
      CALL  "FC41 copy Obj-IF Slave" (
           i_SST_von_Ziel           := #IF_RECEIVER.CONTROL,
           i_SST_an_Ziel            := #IF_RECEIVER.STATUS);
NETWORK
TITLE = FC Rotary valve
      CALL  "FC40 copy Obj-IF Master" (
           i_Freigabe               := #IF_FC_RotaryFeeder.CONTROL.CMD.Request,
           i_Ziel_DB                := #IF_FC_RotaryFeeder_DB,
           i_Ziel_DW                := #IF_FC_RotaryFeeder_DW,
           i_SST_von_Ziel           := #IF_FC_RotaryFeeder.STATUS,
           i_SST_an_Ziel            := #IF_FC_RotaryFeeder.CONTROL,
           Ziel_frei                := #INTERNAL.IF.FC_RotaryValve_ready);
END_FUNCTION_BLOCK

FUNCTION_BLOCK "REC01"	// FB 1011
TITLE = REC01
//Creation:
//Date:            Author:                                               Version
//--------------------------------------------------------------------------------
//14.04.2017     Ilia Bedniakov (ilia)                                   01.00.00
//
//Changes:
//No. Date:        Who       Description                           Mark   Version 
//--------------------------------------------------------------------------------
//01
//________________________________________________________________________________
//Function:
AUTHOR : ilia
VERSION : 0.1
VAR_INPUT
  IF_Blower_DB : INT ;	//Blower DB Nr
  IF_Blower_DW : INT ;	//Receiver Interface Start DW Nr
  iSystemActive : BOOL ;	//system control on
  iSafetySwitchRF_ok : BOOL ;	//safety switch
  iToolKeyControlRF_ok : BOOL ;	//tool control safety swicth
  iSafetySwitchMS_ok : BOOL ;	//safety switch metal separator
  iPFCPM_Ready : BOOL ;	//PFC from Rovema
  iPFCPM_TakeProduct : BOOL ;	//PFC Signal from Rovema
  iRepRotaryFeeder_on : BOOL ;	//repair switch
  iRepScreener_on : BOOL ;	//repair switch
  iRepMetalSeparator_on : BOOL ;	//repair switch
  iFBRotaryFeeder_on : BOOL ;	//FB - feedback
  iFBScreener_on : BOOL ;	//FB - feedback
  iFBMetalSeparator_on : BOOL ;	//FB - feedback
  iHighLevelREC01_free : BOOL ;	//high level sensor
  iLowLevelREC01_free : BOOL ;	//low level sensor
  iHighLevelHP03_free : BOOL ;	//high level sensor
  iLowLevelHP03_free : BOOL ;	//low level sensor
  aRepRotaryValve : BOOL ;	//acknowledge rep. switch fault
  aRepScreener : BOOL ;	//acknowledge rep. switch fault
  aRepMetalSeparator : BOOL ;	//acknowledge rep. switch fault
  aFBRotaryValve : BOOL ;	//acknowledge feedback fault
  aFBScreener : BOOL ;	//acknowledge feedback fault
  aFBMetalSeparator : BOOL ;	//acknowledge feedback fault
  aSafetySwitchRV : BOOL ;
  aToolKeyControlRF : BOOL ;
  aSafetySwitchSM : BOOL ;
  aFullREC01 : BOOL ;
  aSiloNrNotCorrect : BOOL ;	//ak
END_VAR
VAR_IN_OUT
  qRotaryValve_on : BOOL ;	//output signal to motor/valve/FU release
  qScreener_on : BOOL ;	//output signal to motor/valve/FU release
  qMetalSeparator_on : BOOL ;	//output signal to motor/valve/FU release
  qAPBRotaryValve_on : BOOL ;	//output signal to motor/valve/FU release
  qPurgingFilterV1_on : BOOL ;	//output signal to motor/valve/FU release
  qPurgingFilterV2_on : BOOL ;	//output signal to motor/valve/FU release
  qPurgingFilterV3_on : BOOL ;	//output signal to motor/valve/FU release
  qPFCPM_Product : BOOL ;
  qPFCPM_Active : BOOL ;
  fRepRotaryValve : BOOL ;	//Fault
  fRepScreener : BOOL ;	//Fault
  fRepMetalSeparator : BOOL ;	//Fault
  fFBRotaryFeeder : BOOL ;	//Fault
  fFBScreener : BOOL ;	//Fault
  fFBMetalSeparator : BOOL ;	//Fault
  fSafetyRotaryFeeder : BOOL ;	//Fault
  fToolKeyControl : BOOL ;	//Fault
  fSafetyMS : BOOL ;
  fREC01HighLevel : BOOL ;	//Fault
  fHP03HighLevel : BOOL ;
  fREC01_LLCovered : BOOL ;
  fSiloNrNotCorrect : BOOL ;
  fLineNotEmpty : BOOL ;
END_VAR
VAR
  reserve_IO : ARRAY  [12 .. 49 ] OF BYTE ;
  HMI : STRUCT 	//Interface of HMI
   CMD : STRUCT
    StartFeeding : BOOL ;
    REC01_set_empty : BOOL ;	//VISU command button
    HP03_set_empty : BOOL ;
    REC01_disch_forbidden : BOOL ;
    reserve_2 : BOOL ;
    reserve_3 : BOOL ;
    reserve_4 : BOOL ;
    reserve_5 : BOOL ;
    reserve_6 : BOOL ;
    reserve_7 : BOOL ;
    reserve_8 : BOOL ;
    reserve_9 : BOOL ;
    reserve_10 : BOOL ;
    reserve_11 : BOOL ;
    reserve_12 : BOOL ;
    reserve_13 : BOOL ;
   END_STRUCT ;
   STATE : STRUCT
    REC01_empty : BOOL ;
    REC01_full : BOOL ;
    HP03_empty : BOOL ;
    HP03_full : BOOL ;
    REC01_material_signal : BOOL ;
    HP03_material_signal : BOOL ;
    cleaning_active : BOOL ;
    ChangingHpBlocked : BOOL ;
    FROMRovemaReady : BOOL ;
    FROMRovemaTakeMaterial : BOOL ;
    TORovemaProductHP03 : BOOL ;
    TORovemaActive : BOOL ;
    reserve : BOOL ;
    reserve_11 : BOOL ;
    reserve_12 : BOOL ;
    reserve_13 : BOOL ;
   END_STRUCT ;
   PARAM : STRUCT
    PressureBuildTime : REAL  := 3.000000e+000;	//pressure building time
    DelayScreener : REAL  := 1.000000e+001;	//Off delay for screener time
    DelayLowLevelREC01 : REAL  := 3.000000e+001;	//after this time and not free LL sensor stop filling
    DelayFillingExceeded : REAL ;	//no new material + empty pressure -> warning
    CleaningDuration : REAL  := 1.500000e+001;	//cleaning pipeline dutration
    RestDischargeREC01 : REAL  := 2.000000e+001;	//rd for REC01
    RestDischargeHP03 : REAL  := 2.000000e+001;	//rd for HP03
    DelayHighLevelHP03 : REAL  := 5.000000e+000;	//after enclosing HL sensor HP03 delay for discharg starts again
    StorageLocation : INT ;	//Set storage location HP01/HP02
    reserve_7 : INT ;
    reserve_8 : INT ;
    reserve_9 : INT ;
    reserve_10 : INT ;
    reserve_11 : INT ;
   END_STRUCT ;
   PV : STRUCT
    PressureBuildTime : REAL ;
    DelayScreener : REAL ;
    DelayLowLevelREC01 : REAL ;
    DelayFillingExceeded : REAL ;
    CleaningDuration : REAL ;
    RestDischargeREC01 : REAL ;
    RestDischargeHP03 : REAL ;
    DelayHP03HighLevel : REAL ;
    reserve_5 : REAL ;
    StorageLocation : INT ;
    StatusProcessFilling : INT ;	//0-Idle, 1-Release Not Active, 2 - Active
    StatusProcessDischarging : INT ;	//0-Idle, 1-Release Not Active, 2 - Active
    reserve_8 : INT ;
    reserve_9 : INT ;
    reserve_10 : INT ;
   END_STRUCT ;
   PROD : STRUCT
    reserve : ARRAY  [1 .. 50 ] OF BYTE ;
   END_STRUCT ;
  END_STRUCT ;
  PROD : STRUCT 	//Interface of Production
   FROM : STRUCT
    reserve : INT ;
    reserve_1 : INT ;
    reserve_2 : INT ;
    reserve_3 : INT ;
    reserve_4 : INT ;
    reserve_5 : REAL ;
    reserve_6 : REAL ;
    CMD : STRUCT
     reserve : BOOL ;
     reserve_1 : BOOL ;
     reserve_2 : BOOL ;
     reserve_3 : BOOL ;
     reserve_4 : BOOL ;
     reserve_5 : BOOL ;
     reserve_6 : BOOL ;
     reserve_7 : BOOL ;
     reserve_8 : BOOL ;
     reserve_9 : BOOL ;
     reserve_10 : BOOL ;
     reserve_11 : BOOL ;
     reserve_12 : BOOL ;
     reserve_13 : BOOL ;
     reserve_14 : BOOL ;
     reserve_15 : BOOL ;
    END_STRUCT ;
   END_STRUCT ;
   TO : STRUCT
    reserve : INT ;
    reserve_1 : INT ;
    reserve_2 : INT ;
    reserve_3 : INT ;
    reserve_4 : INT ;
    reserve_5 : REAL ;
    reserve_6 : REAL ;
    STATE : STRUCT
     reserve : BOOL ;
     reserve_1 : BOOL ;
     reserve_2 : BOOL ;
     reserve_3 : BOOL ;
     reserve_4 : BOOL ;
     reserve_5 : BOOL ;
     reserve_6 : BOOL ;
     reserve_7 : BOOL ;
     reserve_8 : BOOL ;
     reserve_9 : BOOL ;
     reserve_10 : BOOL ;
     reserve_11 : BOOL ;
     reserve_12 : BOOL ;
     reserve_13 : BOOL ;
     reserve_14 : BOOL ;
     reserve_15 : BOOL ;
    END_STRUCT ;
   END_STRUCT ;
   reserve : ARRAY  [40 .. 49 ] OF BYTE ;
  END_STRUCT ;
  reserve_HMI : ARRAY  [246 .. 299 ] OF BYTE ;
  IF_Blower : STRUCT 	//Interface Blower in active object
   STATUS : STRUCT
    reserve_1 : INT ;
    reserve_2 : INT ;
    reserve_3 : INT ;
    reserve_4 : INT ;
    reserve_5 : INT ;
    ActualPressure : REAL ;
    reserve_6 : REAL ;
    STATE : STRUCT
     Ready : BOOL ;
     Active : BOOL ;
     PressureFault : BOOL ;
     EmptyPressure : BOOL ;
     reserve : BOOL ;
     reserve_1 : BOOL ;
     reserve_2 : BOOL ;
     reserve_3 : BOOL ;
     reserve_4 : BOOL ;
     reserve_5 : BOOL ;
     reserve_6 : BOOL ;
     reserve_7 : BOOL ;
     reserve_8 : BOOL ;
     reserve_9 : BOOL ;
     reserve_10 : BOOL ;
     reserve_11 : BOOL ;
    END_STRUCT ;
   END_STRUCT ;
   CONTROL : STRUCT
    Answer_DB : INT ;
    Answer_DW : INT ;
    reserve_1 : INT ;
    reserve_2 : INT ;
    reserve_3 : INT ;
    reserve_4 : REAL ;
    reserve_5 : REAL ;
    CMD : STRUCT
     Request : BOOL ;
     Release : BOOL ;
     REC01_full : BOOL ;
     reserve_1 : BOOL ;
     reserve_2 : BOOL ;
     reserve_3 : BOOL ;
     reserve_4 : BOOL ;
     reserve_5 : BOOL ;
     reserve_6 : BOOL ;
     reserve_7 : BOOL ;
     reserve_8 : BOOL ;
     reserve_9 : BOOL ;
     reserve_10 : BOOL ;
     reserve_11 : BOOL ;
     reserve_12 : BOOL ;
     reserve_13 : BOOL ;
    END_STRUCT ;
   END_STRUCT ;
  END_STRUCT ;
  IF_Silo : STRUCT
   STATUS : STRUCT
    reserve_1 : INT ;
    reserve_2 : INT ;
    reserve_3 : INT ;
    reserve_4 : INT ;
    reserve_5 : INT ;
    ActualPressure : REAL ;
    reserve_6 : REAL ;
    STATE : STRUCT
     Ready : BOOL ;
     Active : BOOL ;
     PressureFault : BOOL ;
     EmptyPressure : BOOL ;
     reserve : BOOL ;
     reserve_1 : BOOL ;
     reserve_2 : BOOL ;
     reserve_3 : BOOL ;
     reserve_4 : BOOL ;
     reserve_5 : BOOL ;
     reserve_6 : BOOL ;
     reserve_7 : BOOL ;
     reserve_8 : BOOL ;
     reserve_9 : BOOL ;
     reserve_10 : BOOL ;
     reserve_11 : BOOL ;
    END_STRUCT ;
   END_STRUCT ;
   CONTROL : STRUCT
    Answer_DB : INT ;
    Answer_DW : INT ;
    reserve_1 : INT ;
    reserve_2 : INT ;
    reserve_3 : INT ;
    reserve_4 : REAL ;
    reserve_5 : REAL ;
    CMD : STRUCT
     Request : BOOL ;
     Release : BOOL ;
     RECFull : BOOL ;
     reserve_1 : BOOL ;
     reserve_2 : BOOL ;
     reserve_3 : BOOL ;
     reserve_4 : BOOL ;
     reserve_5 : BOOL ;
     reserve_6 : BOOL ;
     reserve_7 : BOOL ;
     reserve_8 : BOOL ;
     reserve_9 : BOOL ;
     reserve_10 : BOOL ;
     reserve_11 : BOOL ;
     reserve_12 : BOOL ;
     reserve_13 : BOOL ;
    END_STRUCT ;
   END_STRUCT ;
  END_STRUCT ;
  reserve_IF : ARRAY  [380 .. 499 ] OF BYTE ;
  RotaryFeeder : STRUCT 	//motor object
   parameter : STRUCT
    motor_on : BOOL  := TRUE;	//activate motor structure
    clock_on : BOOL ;	//activate clock structure
    FC_on : BOOL ;	//activate frequency converter structure
    hour_meter_on : BOOL ;	//activate hour meter
    reserve_4 : BOOL ;
    reserve_5 : BOOL ;
    reserve_6 : BOOL ;
    reserve_7 : BOOL ;
   END_STRUCT ;
   quit_motor : BOOL ;	//1 = quit motor on
   input_motor : BOOL ;	//1 = input motor on (return indication)
   motor_locked : BOOL ;	//1 = motor locked (in manual and auto mode) e.g. repair-/safety switch
   auto_mode_control : BOOL ;	//1 = release/control of motor in auto mode
   motor_in_operation : BOOL ;	//1 = signal motor in operation
   fault : BOOL ;	//1 = signal motor fault
   man_mode_to_SCADA : BOOL ;	//0 = Automatik Mode, 1 = Hand Mode
   man_mode_from_SCADA : BOOL ;	//0 = Automatik Mode, 1 = Hand Mode
   man_mode_control : BOOL ;	//1 = release/control of motor in manual mode (from SCADA)
   man_mode_locked : BOOL ;	//1 = change to manual mode locked, motor is in automatic use
   start_with_impulse : BOOL  := TRUE;	//1 = start cycle with impulse
   set_cycles_reached : BOOL ;	//1 = set number of cycles has been reached
   continous_clock : BOOL  := TRUE;	//1 = continous clock / 0 = set number of clocks
   simulation : BOOL ;	//1 = simulation of object
   release_clock : BOOL ;	//1 = release bit for clock FC
   quit_clock : BOOL ;	//quit for clock FC, if release_clock = TRUE
   set_time_fault : INT  := 5;	//fault evaluation time in seconds
   actual_time_fault : INT ;	//actual fault evaluation time in seconds
   impulse_time : REAL  := 5.000000e+000;	//impulse time for clock in seconds
   break_time : REAL  := 5.000000e+000;	//break time for clock in seconds
   time_counter : REAL ;	//time counter (elapsed time)
   set_cycles : INT ;	//number of clocks if not continous clock
   clock_counter : INT ;	//clock counter
   FCs : STRUCT 	//frequency converter
    FC_in_operation : BOOL ;	//1 = FU in Betrieb
    fault : BOOL ;	//1 = FC fault
    set_revolutions_man_mode : INT ;	//revolutions in permille in manual mode
    actual_revolutions : INT ;	//actual revolutions FC in man/auto mode
   END_STRUCT ;
   hour_meter : STRUCT 	//hour meter
    reset : BOOL ;	//reset hour meter
    warning : BOOL ;	//warning time exceeded
    alarm : BOOL ;	//alarm time exceeded
    actual_operating_hours : REAL ;	//actual operating hours (in hours)
    set_time_warning : REAL ;	//set time for warning (in hours)
    set_time_alarm : REAL ;	//set time for alarm (in hours)
    second_counter_oh : INT ;	//seconds of the actual operatin hours
   END_STRUCT ;
   system_on : BOOL ;	//system released resepectively system area released after emergency stopping
   object_state : INT ;	//1=grey; 5=green; 9=white; 15=yellow; 16=red
  END_STRUCT ;
  Screener : STRUCT 	//motor object
   parameter : STRUCT
    motor_on : BOOL  := TRUE;	//activate motor structure
    clock_on : BOOL ;	//activate clock structure
    FC_on : BOOL ;	//activate frequency converter structure
    hour_meter_on : BOOL ;	//activate hour meter
    reserve_4 : BOOL ;
    reserve_5 : BOOL ;
    reserve_6 : BOOL ;
    reserve_7 : BOOL ;
   END_STRUCT ;
   quit_motor : BOOL ;	//1 = quit motor on
   input_motor : BOOL ;	//1 = input motor on (return indication)
   motor_locked : BOOL ;	//1 = motor locked (in manual and auto mode) e.g. repair-/safety switch
   auto_mode_control : BOOL ;	//1 = release/control of motor in auto mode
   motor_in_operation : BOOL ;	//1 = signal motor in operation
   fault : BOOL ;	//1 = signal motor fault
   man_mode_to_SCADA : BOOL ;	//0 = Automatik Mode, 1 = Hand Mode
   man_mode_from_SCADA : BOOL ;	//0 = Automatik Mode, 1 = Hand Mode
   man_mode_control : BOOL ;	//1 = release/control of motor in manual mode (from SCADA)
   man_mode_locked : BOOL ;	//1 = change to manual mode locked, motor is in automatic use
   start_with_impulse : BOOL  := TRUE;	//1 = start cycle with impulse
   set_cycles_reached : BOOL ;	//1 = set number of cycles has been reached
   continous_clock : BOOL  := TRUE;	//1 = continous clock / 0 = set number of clocks
   simulation : BOOL ;	//1 = simulation of object
   release_clock : BOOL ;	//1 = release bit for clock FC
   quit_clock : BOOL ;	//quit for clock FC, if release_clock = TRUE
   set_time_fault : INT  := 5;	//fault evaluation time in seconds
   actual_time_fault : INT ;	//actual fault evaluation time in seconds
   impulse_time : REAL  := 5.000000e+000;	//impulse time for clock in seconds
   break_time : REAL  := 5.000000e+000;	//break time for clock in seconds
   time_counter : REAL ;	//time counter (elapsed time)
   set_cycles : INT ;	//number of clocks if not continous clock
   clock_counter : INT ;	//clock counter
   FCs : STRUCT 	//frequency converter
    FC_in_operation : BOOL ;	//1 = FU in Betrieb
    fault : BOOL ;	//1 = FC fault
    set_revolutions_man_mode : INT ;	//revolutions in permille in manual mode
    actual_revolutions : INT ;	//actual revolutions FC in man/auto mode
   END_STRUCT ;
   hour_meter : STRUCT 	//hour meter
    reset : BOOL ;	//reset hour meter
    warning : BOOL ;	//warning time exceeded
    alarm : BOOL ;	//alarm time exceeded
    actual_operating_hours : REAL ;	//actual operating hours (in hours)
    set_time_warning : REAL ;	//set time for warning (in hours)
    set_time_alarm : REAL ;	//set time for alarm (in hours)
    second_counter_oh : INT ;	//seconds of the actual operatin hours
   END_STRUCT ;
   system_on : BOOL ;	//system released resepectively system area released after emergency stopping
   object_state : INT ;	//1=grey; 5=green; 9=white; 15=yellow; 16=red
  END_STRUCT ;
  MetalSeparator : STRUCT 	//motor object
   parameter : STRUCT
    motor_on : BOOL  := TRUE;	//activate motor structure
    clock_on : BOOL ;	//activate clock structure
    FC_on : BOOL ;	//activate frequency converter structure
    hour_meter_on : BOOL ;	//activate hour meter
    reserve_4 : BOOL ;
    reserve_5 : BOOL ;
    reserve_6 : BOOL ;
    reserve_7 : BOOL ;
   END_STRUCT ;
   quit_motor : BOOL ;	//1 = quit motor on
   input_motor : BOOL ;	//1 = input motor on (return indication)
   motor_locked : BOOL ;	//1 = motor locked (in manual and auto mode) e.g. repair-/safety switch
   auto_mode_control : BOOL ;	//1 = release/control of motor in auto mode
   motor_in_operation : BOOL ;	//1 = signal motor in operation
   fault : BOOL ;	//1 = signal motor fault
   man_mode_to_SCADA : BOOL ;	//0 = Automatik Mode, 1 = Hand Mode
   man_mode_from_SCADA : BOOL ;	//0 = Automatik Mode, 1 = Hand Mode
   man_mode_control : BOOL ;	//1 = release/control of motor in manual mode (from SCADA)
   man_mode_locked : BOOL ;	//1 = change to manual mode locked, motor is in automatic use
   start_with_impulse : BOOL  := TRUE;	//1 = start cycle with impulse
   set_cycles_reached : BOOL ;	//1 = set number of cycles has been reached
   continous_clock : BOOL  := TRUE;	//1 = continous clock / 0 = set number of clocks
   simulation : BOOL ;	//1 = simulation of object
   release_clock : BOOL ;	//1 = release bit for clock FC
   quit_clock : BOOL ;	//quit for clock FC, if release_clock = TRUE
   set_time_fault : INT  := 5;	//fault evaluation time in seconds
   actual_time_fault : INT ;	//actual fault evaluation time in seconds
   impulse_time : REAL  := 5.000000e+000;	//impulse time for clock in seconds
   break_time : REAL  := 5.000000e+000;	//break time for clock in seconds
   time_counter : REAL ;	//time counter (elapsed time)
   set_cycles : INT ;	//number of clocks if not continous clock
   clock_counter : INT ;	//clock counter
   FCs : STRUCT 	//frequency converter
    FC_in_operation : BOOL ;	//1 = FU in Betrieb
    fault : BOOL ;	//1 = FC fault
    set_revolutions_man_mode : INT ;	//revolutions in permille in manual mode
    actual_revolutions : INT ;	//actual revolutions FC in man/auto mode
   END_STRUCT ;
   hour_meter : STRUCT 	//hour meter
    reset : BOOL ;	//reset hour meter
    warning : BOOL ;	//warning time exceeded
    alarm : BOOL ;	//alarm time exceeded
    actual_operating_hours : REAL ;	//actual operating hours (in hours)
    set_time_warning : REAL ;	//set time for warning (in hours)
    set_time_alarm : REAL ;	//set time for alarm (in hours)
    second_counter_oh : INT ;	//seconds of the actual operatin hours
   END_STRUCT ;
   system_on : BOOL ;	//system released resepectively system area released after emergency stopping
   object_state : INT ;	//1=grey; 5=green; 9=white; 15=yellow; 16=red
  END_STRUCT ;
  AirPurgedBearing : STRUCT 	//valve object with 1Q and 0-2I
   parameter : STRUCT
    valve_on : BOOL  := TRUE;	//activate valve structure
    clock_on : BOOL ;	//activate clock structure
    reserve_3 : BOOL ;
    switching_number_on : BOOL ;	//activate switching number counter
    reserve_4 : BOOL ;
    parameter_1Q : BOOL  := TRUE;	//valve type with 1 quit 0 inputs
    parameter_1Q_1I : BOOL ;	//valve type with 1 quit 1 input (=)
    parameter_1Q_1IN : BOOL ;	//valve type with 1 quit 1 input (<>)
    parameter_1Q_2I : BOOL ;	//valve type with 1 quit 2 inputs
    parameter_text_pos_1 : BOOL ;
    parameter_text_straight : BOOL ;
    parameter_text_inverse : BOOL ;	//select text inverse = "close/open" or "bypass/convey" aso.
    parameter_text_open : BOOL ;	//select text quit = "open/close"
    parameter_text_convey : BOOL ;	//select text quit = "convey/bypass"
    parameter_text_on : BOOL  := TRUE;	//select text quit = "on/off"
    parameter_text_up : BOOL ;	//select text quit = "up/down"
   END_STRUCT ;
   quit_valve : BOOL ;	//1 = quit valve
   input_valve_set : BOOL ;	//1 = input valve, if quit valve set
   input_valve_not_set : BOOL ;	//1 = input valve, if quit valve not set
   auto_mode_control : BOOL ;	//1 = release/control of valve in auto mode
   valve_in_operation : BOOL ;	//1 = signal valve in operation
   fault : BOOL ;	//1 = signal valve fault
   man_mode_to_SCADA : BOOL ;	//0 = automatic mode , 1 = manual mode
   man_mode_from_SCADA : BOOL ;	//0 = automatic mode , 1 = manual mode
   man_mode_control : BOOL ;	//1 = release/control of valve in manual mode (from SCADA)
   man_mode_locked : BOOL ;	//1 = change to manual mode locked, valve is in automatic use
   start_with_impulse : BOOL ;	//1 = start cycle with impluse
   set_cycles_reached : BOOL ;	//1 = set number of cycles has been reached
   continous_clock : BOOL ;	//1 = continous clock / 0 = set number of clocks
   simulation : BOOL ;	//1 = simulation of object
   release_clock : BOOL ;	//1 = release bit for clock FC
   quit_clock : BOOL ;	//quit for clock FC, if release_clock = TRUE
   set_time_fault : INT  := 5;	//fault evaluation time in seconds
   actual_time_fault : INT ;	//actual fault evaluation time in seconds
   impulse_time : REAL  := 5.000000e+000;	//impulse time for clock in seconds
   break_time : REAL  := 5.000000e+000;	//break time for clock in seconds
   time_counter : REAL ;	//time counter (elapsed time)
   set_cycles : INT ;	//number of clocks if not continous clock
   clock_counter : INT ;	//clock counter
   switching_number_counter : STRUCT 	//switching number counter
    reset : BOOL ;	//reset switching number counter
    warning : BOOL ;	//warning number exceeded
    alarm : BOOL ;	//alarm number exceeded
    flank_flag : BOOL ;	//internal flag
    actual_switching_number : REAL ;	//actual switching number
    set_number_warning : REAL ;	//set number for warning
    set_number_alarm : REAL ;	//set number for alarm
   END_STRUCT ;
   set_time_in_operation : INT ;	//1IoO: set time for delay of "valve in operation"
   real_time_in_operation : INT ;	//1IoO: real time for delay of "valve in operation"
   system_on : BOOL ;	//system released resepectively system area released after emergency stopping
   reserve : ARRAY  [44 .. 47 ] OF BYTE ;
   object_state : INT ;	//1=grey; 5=green; 9=white; 15=yellow; 16=red
  END_STRUCT ;
  PurgedFilter : STRUCT 	//valve object with 1-10 quits with clock (e.g. filter cleaning)
   parameter : STRUCT
    valve_on : BOOL  := TRUE;	//activate valve structure
    clock_1_on : BOOL  := TRUE;	//activate clock structure 1
    clock_2_on : BOOL  := TRUE;	//activate clock structure 2
    switching_number_on : BOOL ;	//activate switching number counter
    hour_meter_on : BOOL ;	//activate hour meter
    reserve_5 : BOOL ;
    reserve_6 : BOOL ;
    reserve_7 : BOOL ;
    reserve_8 : BOOL ;
    reserve_9 : BOOL ;
    reserve_10 : BOOL ;
    reserve_11 : BOOL ;
    reserve_12 : BOOL ;
    reserve_13 : BOOL ;
    reserve_14 : BOOL ;
    reserve_15 : BOOL ;
   END_STRUCT ;
   quit_valve_1 : BOOL ;	//1 = quit valve 1
   quit_valve_2 : BOOL ;	//1 = quit valve 2
   quit_valve_3 : BOOL ;	//1 = quit valve 3
   quit_valve_4 : BOOL ;	//1 = quit valve 4
   quit_valve_5 : BOOL ;	//1 = quit valve 5
   quit_valve_6 : BOOL ;	//1 = quit valve 6
   quit_valve_7 : BOOL ;	//1 = quit valve 7
   quit_valve_8 : BOOL ;	//1 = quit valve 8
   quit_valve_9 : BOOL ;	//1 = quit valve 9
   quit_valve_10 : BOOL ;	//1 = quit valve 10
   auto_mode_control_clock1 : BOOL ;	//1 = release/control valve with clock 1 in auto mode
   auto_mode_control_clock2 : BOOL ;	//1 = release/control valve with clock 2 in auto mode
   valve_in_operation : BOOL ;	//1 = signal valve/valves in operation
   man_mode_to_SCADA : BOOL ;	//0 = automatic mode , 1 = manual mode
   man_mode_from_SCADA : BOOL ;	//0 = automatic mode , 1 = manual mode
   man_mode_control_valve_1 : BOOL ;	//1 = release/control valve 1 in manual mode (from SCADA)
   man_mode_control_valve_2 : BOOL ;	//1 = release/control valve 2 in manual mode (from SCADA)
   man_mode_control_valve_3 : BOOL ;	//1 = release/control valve 3 in manual mode (from SCADA)
   man_mode_control_valve_4 : BOOL ;	//1 = release/control valve 4 in manual mode (from SCADA)
   man_mode_control_valve_5 : BOOL ;	//1 = release/control valve 5 in manual mode (from SCADA)
   man_mode_control_valve_6 : BOOL ;	//1 = release/control valve 6 in manual mode (from SCADA)
   man_mode_control_valve_7 : BOOL ;	//1 = release/control valve 7 in manual mode (from SCADA)
   man_mode_control_valve_8 : BOOL ;	//1 = release/control valve 8 in manual mode (from SCADA)
   man_mode_control_valve_9 : BOOL ;	//1 = release/control valve 9 in manual mode (from SCADA)
   man_mode_contrl_valve_10 : BOOL ;	//1 = release/control valve 10 in manual mode (from SCADA)
   man_mode_locked : BOOL ;	//1 = change to manual mode locked, valve is in automatic use
   start_with_impulse : BOOL  := TRUE;	//1 = start cycle with impluse
   set_cycles_reached : BOOL ;	//1 = set number of cycles has been reached
   continous_clock : BOOL  := TRUE;	//1 = continous clock / 0 = set number of clocks
   system_on : BOOL ;	//system released resepectively system area released after emergency stopping
   impulse_time_filling : REAL  := 5.000000e-001;	//impulse time for filling clock in seconds (clock 1)
   break_time_filling : REAL  := 3.000000e+001;	//break time for filling clock in seconds (clock 1)
   impulse_time_discharge : REAL  := 5.000000e-001;	//impulse time for discharge clock in seconds (clock 2)
   break_time_discharge : REAL  := 1.000000e+001;	//break time for discharge clock in seconds (clock 2)
   time_counter : REAL ;	//time counter (elapsed time)
   set_cycles : INT ;	//number of clocks if not continous clock
   clock_counter : INT ;	//clock counter
   number_of_valves : INT  := 3;	//number of used valves
   switching_number_counter : STRUCT 	//switching number counter / hour meter
    reset : BOOL ;	//reset switching number counter / hour meter
    warning : BOOL ;	//warning number / time exceeded
    alarm : BOOL ;	//alarm number / time exceeded
    flank_flag : BOOL ;	//internal flag
    release_counter : BOOL ;	//release switching number counter / hour meter
    actual_switching_number : REAL ;	//actual switching number / hour meter
    set_number_warning : REAL ;	//set number / time for warning
    set_number_alarm : REAL ;	//set number / time for alarm
   END_STRUCT ;
   reserve1 : ARRAY  [46 .. 47 ] OF BYTE ;
   object_state : INT ;	//1=grey; 5=green; 15=yellow
  END_STRUCT ;
  LevelIndicators : STRUCT
   HighLevelREC01 : STRUCT
    input : BOOL ;
    debounced_covered : BOOL ;
    helpmarker : BOOL ;
    Fehler : BOOL ;
   END_STRUCT ;
   LowLevelREC01 : STRUCT
    input : BOOL ;
    debounced_covered : BOOL ;
    helpmarker : BOOL ;
    fault : BOOL ;
   END_STRUCT ;
   HighLevelHP03 : STRUCT
    input : BOOL ;
    debounced_covered : BOOL ;
    helpmarker : BOOL ;
    Fehler : BOOL ;
   END_STRUCT ;
   LowLevelHP03 : STRUCT
    input : BOOL ;
    debounced_covered : BOOL ;
    helpmarker : BOOL ;
    Fehler : BOOL ;
   END_STRUCT ;
  END_STRUCT ;
  reserve_Cmod : ARRAY  [758 .. 849 ] OF BYTE ;
  TIMERS : STRUCT 	//ten timers
   TON_REC01_RestDischarge : STRUCT
    IN : BOOL ;
    RST : BOOL ;
    IMP : BOOL ;
    Q : BOOL ;
    PT : REAL ;
    ET : REAL ;
   END_STRUCT ;
   TON_HP03_RestDischarge : STRUCT
    IN : BOOL ;
    RST : BOOL ;
    IMP : BOOL ;
    Q : BOOL ;
    PT : REAL ;
    ET : REAL ;
   END_STRUCT ;
   XX_TON_PressureBuildTime : STRUCT
    IN : BOOL ;
    RST : BOOL ;
    IMP : BOOL ;
    Q : BOOL ;
    PT : REAL ;
    ET : REAL ;
   END_STRUCT ;
   TOF_MetalSeparator_Delay : STRUCT
    IN : BOOL ;
    RST : BOOL ;
    IMP : BOOL ;
    Q : BOOL ;
    PT : REAL ;
    ET : REAL ;
   END_STRUCT ;
   TOF_Screener_Delay : STRUCT
    IN : BOOL ;
    RST : BOOL ;
    IMP : BOOL ;
    Q : BOOL ;
    PT : REAL ;
    ET : REAL ;
   END_STRUCT ;
   TOF_AirPurgedBearing : STRUCT
    IN : BOOL ;
    RST : BOOL ;
    IMP : BOOL ;
    Q : BOOL ;
    PT : REAL ;
    ET : REAL ;
   END_STRUCT ;
   TON_HP03_HL_DISCLOSURE : STRUCT
    IN : BOOL ;
    RST : BOOL ;
    IMP : BOOL ;
    Q : BOOL ;
    PT : REAL ;
    ET : REAL ;
   END_STRUCT ;
   TON_REC01_LowLevCovered : STRUCT
    IN : BOOL ;
    RST : BOOL ;
    IMP : BOOL ;
    Q : BOOL ;
    PT : REAL ;
    ET : REAL ;
   END_STRUCT ;
   TV_CleaningLineDuration : STRUCT
    IN : BOOL ;
    RST : BOOL ;
    IMP : BOOL ;
    Q : BOOL ;
    PT : REAL ;
    ET : REAL ;
   END_STRUCT ;
   TON_HighLevel_blocked : STRUCT 	//// ak
    IN : BOOL ;
    RST : BOOL ;
    IMP : BOOL ;
    Q : BOOL ;
    PT : REAL ;
    ET : REAL ;
   END_STRUCT ;
   reserve_1 : STRUCT
    IN : BOOL ;
    RST : BOOL ;
    IMP : BOOL ;
    Q : BOOL ;
    PT : REAL ;
    ET : REAL ;
   END_STRUCT ;
  END_STRUCT ;
  SEQUENCE : STRUCT
   Filling : STRUCT
    AUTO : BOOL ;
    MANUAL : BOOL ;
    LOCKED : BOOL ;
    RELEASE : BOOL ;
    ACTIVE : BOOL ;
    reserve_2 : BOOL ;
    reserve_3 : BOOL ;
    reserve_4 : BOOL ;
    reserve_5 : BOOL ;
    reserve_6 : BOOL ;
    reserve_7 : BOOL ;
    reserve_8 : BOOL ;
    reserve_9 : BOOL ;
    reserve_10 : BOOL ;
    reserve_11 : BOOL ;
    reserve_12 : BOOL ;
   END_STRUCT ;
   Discharging : STRUCT
    AUTO : BOOL ;
    MANUAL : BOOL ;
    LOCKED : BOOL ;
    RELEASE : BOOL ;
    ACTIVE : BOOL ;
    reserve_2 : BOOL ;
    reserve_3 : BOOL ;
    reserve_4 : BOOL ;
    reserve_5 : BOOL ;
    reserve_6 : BOOL ;
    reserve_7 : BOOL ;
    reserve_8 : BOOL ;
    reserve_9 : BOOL ;
    reserve_10 : BOOL ;
    reserve_11 : BOOL ;
    reserve_12 : BOOL ;
   END_STRUCT ;
   reserve : ARRAY  [4 .. 99 ] OF BYTE ;
  END_STRUCT ;
  INTERNAL : STRUCT
   IF : STRUCT
    Silo : STRUCT
     StorageLocationNumber : INT ;
     StorageLocation_DB : INT ;
     StorageLocation_DW : INT ;
     reserve : INT ;
     Silo_ready : BOOL ;
     Silo_free : BOOL ;
     SiloNr_correct : BOOL ;
     reserve_3_2 : BOOL ;
     reserve_1_1 : BOOL ;
     reserve_2_1 : BOOL ;
     reserve_3_1 : BOOL ;
     reserve_3_1_1 : BOOL ;
     reserve_1 : INT ;
     reserve_2 : INT ;
     reserve_3 : INT ;
    END_STRUCT ;
    Blower : STRUCT
     Blower_DB : INT ;
     Blower_DW : INT ;
     reserve : INT ;
     Blower_ready : BOOL ;
     Blower_free : BOOL ;
     reserve_2 : BOOL ;
     reserve_3 : BOOL ;
     reserve_1_1 : BOOL ;
     reserve_2_1 : BOOL ;
     reserve_3_1 : BOOL ;
     reserve_3_1_1 : BOOL ;
    END_STRUCT ;
    reserve_5 : BOOL ;
    reserve_6 : BOOL ;
    reserve_7 : BOOL ;
    reserve_8 : BOOL ;
    reserve_9 : BOOL ;
    reserve_10 : BOOL ;
    reserve_11 : BOOL ;
    reserve_12 : BOOL ;
   END_STRUCT ;
   Flags : STRUCT
    xx_FP_Material_REC01 : STRUCT
     helpBit : BOOL ;
     pulseBit : BOOL ;
    END_STRUCT ;
    xx_FP_Material_HP03 : STRUCT
     helpBit : BOOL ;
     pulseBit : BOOL ;
    END_STRUCT ;
    FP_releaseFilling : STRUCT
     helpBit : BOOL ;
     pulseBit : BOOL ;
    END_STRUCT ;
    FP_StorageLocReset : STRUCT
     helpBit : BOOL ;
     pulseBit : BOOL ;
    END_STRUCT ;
    XX_FP_CleaningFinished : STRUCT
     helpBit : BOOL ;
     pulseBit : BOOL ;
    END_STRUCT ;
    FP_Start_wo_Silocorrect : STRUCT
     helpBit : BOOL ;
     pulseBit : BOOL ;
    END_STRUCT ;
    FP_CleaningRelease : STRUCT
     helpBit : BOOL ;
     pulseBit : BOOL ;
    END_STRUCT ;
    StatusREC01 : STRUCT
     REC01_empty : BOOL ;
     REC01_full : BOOL ;
     REC01_LowLevelCovered : BOOL ;
     REC01_material_signal : BOOL ;
     reserve_1 : BOOL ;
     reserve_2 : BOOL ;
     reserve_3 : BOOL ;
     reserve_4 : BOOL ;
    END_STRUCT ;
    StatusHP03 : STRUCT
     HP03_empty : BOOL ;
     HP03_full : BOOL ;
     HP03_HL_disclosured : BOOL ;
     HP03_material_signal : BOOL ;
     filling_locked : BOOL ;
     reserve_2 : BOOL ;
     reserve_3 : BOOL ;
     reserve_4 : BOOL ;
    END_STRUCT ;
    reserve_1 : STRUCT
     HP03_empty : BOOL ;
     HP03_full : BOOL ;
     HP03_HL_disclosured : BOOL ;
     HP03_material_signal : BOOL ;
     reserve_1 : BOOL ;
     reserve_2 : BOOL ;
     reserve_3 : BOOL ;
     reserve_4 : BOOL ;
    END_STRUCT ;
    ReleaseFeeding : BOOL ;
    reserve_2 : BOOL ;
    CleaningRelease : BOOL ;
    CleaningFinished : BOOL ;
    DischargeREC01_forbidden : BOOL ;
    reserve : BOOL ;
    reserve_4 : BOOL ;
    reserve_6 : BOOL ;
   END_STRUCT ;
   Instance_DB_number : INT ;
  END_STRUCT ;
END_VAR
VAR_TEMP
  StorageLoc_List_DW : INT ;
  StorageLocCopyError : INT ;
  tempDB : INT ;
END_VAR
BEGIN
NETWORK
TITLE = ---- instance DB ----
      L     0;
      L     DINO;
      ==I;
      BEC;
      T     #INTERNAL.Instance_DB_number;
NETWORK
TITLE = ------------------------ Sensors------------------------- 
NETWORK
TITLE = REC01 Low Level Sensor
      AN    #iLowLevelREC01_free;
      =     #LevelIndicators.LowLevelREC01.input;
      CALL  "FC14 Debounce Indicator" (
           Eingang                  := #LevelIndicators.LowLevelREC01.input,
           Takt                     := "M 1.6 ClckDdebounceIndic",
           Folgemerker              := #LevelIndicators.LowLevelREC01.helpmarker,
           Eingang_entprellt        := #LevelIndicators.LowLevelREC01.debounced_covered);
NETWORK
TITLE = REC01 Low Level Sensor Covered TOF Delay
      AN    #iLowLevelREC01_free;
      AN    #fREC01HighLevel;	// ak
      A(;	// ak
      O     #RotaryFeeder.motor_in_operation;	// ak
      O     #RotaryFeeder.man_mode_from_SCADA;	// ak
      );	// ak
      =     #TIMERS.TON_REC01_LowLevCovered.IN;
      CALL  "FC3 Cycle generator" (
           in_Freigabe              := #TIMERS.TON_REC01_LowLevCovered.IN,
           in_Reset                 := #TIMERS.TON_REC01_LowLevCovered.RST,
           in_Impuls                := "M 1.7 Cycle Timer-FC",
           in_Impulszeit_in_100ms   := "MW 6 Timer Val Cycle FCs",
           in_Verzoegerungsart      := B#16#45,
           in_Verzoegerungszeit     := #HMI.PARAM.DelayLowLevelREC01,
           io_Ausgangssignal        := #TIMERS.TON_REC01_LowLevCovered.Q,
           io_Zeitzaehler           := #TIMERS.TON_REC01_LowLevCovered.ET);
      L     #TIMERS.TON_REC01_LowLevCovered.ET;
      T     #HMI.PV.DelayLowLevelREC01;
      A     #TIMERS.TON_REC01_LowLevCovered.Q;
      =     #INTERNAL.Flags.StatusREC01.REC01_LowLevelCovered;
      =     #fREC01_LLCovered;
NETWORK
TITLE = REC01 High Level Sensor
      AN    #iHighLevelREC01_free;
      =     #LevelIndicators.HighLevelREC01.input;
      CALL  "FC14 Debounce Indicator" (
           Eingang                  := #LevelIndicators.HighLevelREC01.input,
           Takt                     := "M 4.7 Imp Cycle 2,0-sec",
           Folgemerker              := #LevelIndicators.HighLevelREC01.helpmarker,
           Eingang_entprellt        := #LevelIndicators.HighLevelREC01.debounced_covered);
      A     #LevelIndicators.HighLevelREC01.debounced_covered;
      S     #fREC01HighLevel;
      AN    #LevelIndicators.HighLevelREC01.debounced_covered;
      A     #aFullREC01;
      R     #fREC01HighLevel;
      A     #fREC01HighLevel;
      =     #IF_Silo.CONTROL.CMD.RECFull;
NETWORK
TITLE = HP03 Low Level Sensor
      AN    #iLowLevelHP03_free;
      =     #LevelIndicators.LowLevelHP03.input;
      CALL  "FC14 Debounce Indicator" (
           Eingang                  := #LevelIndicators.LowLevelHP03.input,
           Takt                     := "M 1.6 ClckDdebounceIndic",
           Folgemerker              := #LevelIndicators.LowLevelHP03.helpmarker,
           Eingang_entprellt        := #LevelIndicators.LowLevelHP03.debounced_covered);
NETWORK
TITLE = HP03 High Level Sensor
      AN    #iHighLevelHP03_free;
      =     #LevelIndicators.HighLevelHP03.input;
      CALL  "FC14 Debounce Indicator" (
           Eingang                  := #LevelIndicators.HighLevelHP03.input,
           Takt                     := "M 1.6 ClckDdebounceIndic",
           Folgemerker              := #LevelIndicators.HighLevelHP03.helpmarker,
           Eingang_entprellt        := #LevelIndicators.HighLevelHP03.debounced_covered);
      A     #LevelIndicators.HighLevelHP03.debounced_covered;	// ak
      AN    #RotaryFeeder.motor_in_operation;	// ak
      A     #iPFCPM_TakeProduct;	// ak
      =     #TIMERS.TON_HighLevel_blocked.IN;	// ak
      L     #HMI.PARAM.DelayHighLevelHP03;	// ak
      L     1.500000e+01;
      +R;
      T     #TIMERS.TON_HighLevel_blocked.PT;	// ak
// ak
      CALL  "FC3 Cycle generator" (
           in_Freigabe              := #TIMERS.TON_HighLevel_blocked.IN,
           in_Reset                 := FALSE,
           in_Impuls                := "M 1.7 Cycle Timer-FC",
           in_Impulszeit_in_100ms   := "MW 6 Timer Val Cycle FCs",
           in_Verzoegerungsart      := B#16#45,
           in_Verzoegerungszeit     := #TIMERS.TON_HighLevel_blocked.PT,
           io_Ausgangssignal        := #TIMERS.TON_HighLevel_blocked.Q,
           io_Zeitzaehler           := #TIMERS.TON_HighLevel_blocked.ET);
      A     #LevelIndicators.HighLevelHP03.debounced_covered;
      AN    #LevelIndicators.LowLevelHP03.debounced_covered;	// ak
      O;	//                        ak
      A     #TIMERS.TON_HighLevel_blocked.Q;	//                 ak
      =     #fHP03HighLevel;
NETWORK
TITLE = REC01 intern statuses(material and empty)
      A     #LevelIndicators.LowLevelREC01.debounced_covered;
      A     #LevelIndicators.HighLevelREC01.debounced_covered;
      =     #INTERNAL.Flags.StatusREC01.REC01_full;
      A     #SEQUENCE.Filling.AUTO;
      A(;
      O     #LevelIndicators.LowLevelREC01.debounced_covered;
      O     #LevelIndicators.HighLevelREC01.debounced_covered;
      O;
      A     #IF_Blower.STATUS.STATE.Active;
      A     #IF_Silo.STATUS.STATE.Active;
      );
      S     #INTERNAL.Flags.StatusREC01.REC01_material_signal;
      A     #INTERNAL.Flags.StatusREC01.REC01_material_signal;
      AN    #LevelIndicators.LowLevelREC01.debounced_covered;
      AN    #LevelIndicators.HighLevelREC01.debounced_covered;
      A     #SEQUENCE.Discharging.ACTIVE;
      AN    #IF_Blower.STATUS.STATE.Active;
      AN    #IF_Silo.STATUS.STATE.Active;
      =     #TIMERS.TON_REC01_RestDischarge.IN;
      CALL  "FC3 Cycle generator" (
           in_Freigabe              := #TIMERS.TON_REC01_RestDischarge.IN,
           in_Reset                 := FALSE,
           in_Impuls                := "M 1.7 Cycle Timer-FC",
           in_Impulszeit_in_100ms   := "MW 6 Timer Val Cycle FCs",
           in_Verzoegerungsart      := B#16#45,
           in_Verzoegerungszeit     := #HMI.PARAM.RestDischargeREC01,
           io_Ausgangssignal        := #TIMERS.TON_REC01_RestDischarge.Q,
           io_Zeitzaehler           := #TIMERS.TON_REC01_RestDischarge.ET);
      A     #TIMERS.TON_REC01_RestDischarge.Q;
      O;
      A     #HMI.CMD.REC01_set_empty;	// from VISU
      AN    #LevelIndicators.LowLevelREC01.debounced_covered;
      AN    #LevelIndicators.HighLevelREC01.debounced_covered;
      AN    #SEQUENCE.Filling.ACTIVE;
      AN    #HMI.STATE.cleaning_active;
      R     #INTERNAL.Flags.StatusREC01.REC01_material_signal;
      L     #TIMERS.TON_REC01_RestDischarge.ET;
      T     #HMI.PV.RestDischargeREC01;
      AN    #INTERNAL.Flags.StatusREC01.REC01_material_signal;
      =     #INTERNAL.Flags.StatusREC01.REC01_empty;
NETWORK
TITLE = HP03 intern statuses (material and empty)
// after rest discharge - > EMPTY Status
      A     #LevelIndicators.LowLevelHP03.debounced_covered;
      A     #LevelIndicators.HighLevelHP03.debounced_covered;
      =     #INTERNAL.Flags.StatusHP03.HP03_full;
      A     #SEQUENCE.Discharging.AUTO;
      A(;
      O     #LevelIndicators.LowLevelHP03.debounced_covered;
      O     #LevelIndicators.HighLevelHP03.debounced_covered;
      O;
      A     #RotaryFeeder.motor_in_operation;
      A     #INTERNAL.Flags.StatusREC01.REC01_material_signal;	// ilia
      );
      S     #INTERNAL.Flags.StatusHP03.HP03_material_signal;
      A     #INTERNAL.Flags.StatusHP03.HP03_material_signal;
      AN    #LevelIndicators.LowLevelHP03.debounced_covered;
      AN    #LevelIndicators.HighLevelHP03.debounced_covered;
      A(;
//      AN    #SEQUENCE.Discharging.RELEASE
      AN    #HMI.STATE.cleaning_active;
      A     #iPFCPM_TakeProduct;
      A(;	// ak
      A     #INTERNAL.Flags.StatusREC01.REC01_empty;
      ON    #RotaryFeeder.motor_in_operation;	// ak 
      );
      );
      =     #TIMERS.TON_HP03_RestDischarge.IN;
      CALL  "FC3 Cycle generator" (
           in_Freigabe              := #TIMERS.TON_HP03_RestDischarge.IN,
           in_Reset                 := #TIMERS.TON_HP03_RestDischarge.RST,
           in_Impuls                := "M 1.7 Cycle Timer-FC",
           in_Impulszeit_in_100ms   := "MW 6 Timer Val Cycle FCs",
           in_Verzoegerungsart      := B#16#45,
           in_Verzoegerungszeit     := #HMI.PARAM.RestDischargeHP03,
           io_Ausgangssignal        := #TIMERS.TON_HP03_RestDischarge.Q,
           io_Zeitzaehler           := #TIMERS.TON_HP03_RestDischarge.ET);
      A     #TIMERS.TON_HP03_RestDischarge.Q;
      O;
      A     #HMI.CMD.HP03_set_empty;	// from VISU
      AN    #LevelIndicators.LowLevelHP03.debounced_covered;
      AN    #LevelIndicators.HighLevelHP03.debounced_covered;
      AN    #SEQUENCE.Discharging.RELEASE;
      R     #INTERNAL.Flags.StatusHP03.HP03_material_signal;
      L     #TIMERS.TON_HP03_RestDischarge.ET;
      T     #HMI.PV.RestDischargeHP03;
      AN    #INTERNAL.Flags.StatusHP03.HP03_material_signal;
      =     #INTERNAL.Flags.StatusHP03.HP03_empty;
NETWORK
TITLE = ---- Sequence status ----
NETWORK
TITLE = Sequence filling auto
      AN    #SEQUENCE.Filling.LOCKED;
      =     #SEQUENCE.Filling.AUTO;
NETWORK
TITLE = Sequence filling manual
      O     #PurgedFilter.man_mode_to_SCADA;
      AN    #SEQUENCE.Filling.AUTO;
      =     #SEQUENCE.Filling.MANUAL;
NETWORK
TITLE = Sequence filling locked
      AN    #iSystemActive;
      =     #SEQUENCE.Filling.LOCKED;
NETWORK
TITLE = Sequence discharging auto
      AN    #SEQUENCE.Discharging.LOCKED;
      =     #SEQUENCE.Discharging.AUTO;
NETWORK
TITLE = Sequence discharging manual
      O     #RotaryFeeder.man_mode_to_SCADA;
      O     #Screener.man_mode_to_SCADA;
      O     #MetalSeparator.man_mode_to_SCADA;
      O     #AirPurgedBearing.man_mode_to_SCADA;
      O     #PurgedFilter.man_mode_to_SCADA;
      AN    #SEQUENCE.Discharging.AUTO;
      =     #SEQUENCE.Discharging.MANUAL;
NETWORK
TITLE = Sequence discharging locked
      O     #SEQUENCE.Discharging.MANUAL;
      ON    #iSystemActive;
      O     #fSafetyRotaryFeeder;
      O     #fToolKeyControl;
      O     #fSafetyMS;
      =     #SEQUENCE.Discharging.LOCKED;
NETWORK
TITLE = Set/Reset Release Feeding 
      A     #HMI.CMD.StartFeeding;
      A     #iSystemActive;
      AN    #fSiloNrNotCorrect;
      S     #INTERNAL.Flags.ReleaseFeeding;
      ON    #iSystemActive;
      ON    #HMI.CMD.StartFeeding;
      R     #INTERNAL.Flags.ReleaseFeeding;
//      ON    #iSystemActive  ak
      O     #fSiloNrNotCorrect;
      R     #HMI.CMD.StartFeeding;
NETWORK
TITLE = ---- General status (rep.switches etc.)----
NETWORK
TITLE = RV Tool sensor control
//safety switch
      A     #iToolKeyControlRF_ok;
      A     #aToolKeyControlRF;
      R     #fToolKeyControl;
      AN    #iToolKeyControlRF_ok;
      S     #fToolKeyControl;
NETWORK
TITLE = Rotary valve safety switch and repair switch Faults
//safety switch
      A     #iSafetySwitchRF_ok;
      A     #aSafetySwitchRV;
      R     #fSafetyRotaryFeeder;
      AN    #iSafetySwitchRF_ok;
      S     #fSafetyRotaryFeeder;
//repair switch
      A     #iRepRotaryFeeder_on;
      A     #aRepRotaryValve;
      R     #fRepRotaryValve;
      O     #RotaryFeeder.auto_mode_control;
      O     #RotaryFeeder.man_mode_control;
      AN    #iRepRotaryFeeder_on;
      S     #fRepRotaryValve;
NETWORK
TITLE = Metal Separator (MS) safety switch and repair switch Fault
//safety switch
      A     #iSafetySwitchMS_ok;
      A     #aSafetySwitchSM;
      R     #fSafetyMS;
      AN    #iSafetySwitchMS_ok;
      S     #fSafetyMS;
//repairSwitch
      A     #iRepScreener_on;
      A     #aRepScreener;
      R     #fRepScreener;
      O     #Screener.auto_mode_control;
      O     #Screener.man_mode_control;
      AN    #iRepScreener_on;
      S     #fRepScreener;
NETWORK
TITLE = Metal separator repair switch fault
      A     #iRepMetalSeparator_on;
      A     #aRepMetalSeparator;
      R     #fRepMetalSeparator;
      O     #MetalSeparator.auto_mode_control;
      O     #MetalSeparator.man_mode_control;
      AN    #iRepMetalSeparator_on;
      S     #fRepMetalSeparator;
NETWORK
TITLE = --------------------- Sequence Filling -------------------------
NETWORK
TITLE = Filling: Storage Location from HMI
      A     #iSystemActive;
      AN    #SEQUENCE.Filling.RELEASE;
      AN    #SEQUENCE.Discharging.RELEASE;
      A     #INTERNAL.Flags.StatusHP03.HP03_empty;
      A     #INTERNAL.Flags.StatusREC01.REC01_empty;
      A(;
      L     #HMI.PARAM.StorageLocation;
      L     0;
      <>I;
      );
      A(;
      L     #HMI.PARAM.StorageLocation;
      L     #HMI.PV.StorageLocation;
      <>I;
      );
      JCN   NPA;	// no transport active (dsch or fill)
      L     #HMI.PARAM.StorageLocation;
      T     #HMI.PV.StorageLocation;
NPA:  NOP   0;
NETWORK
TITLE = Filling: Silo number is correct
      O(;
      L     #HMI.PV.StorageLocation;
      L     1;
      ==I;
      );
      O(;
      L     #HMI.PV.StorageLocation;
      L     2;
      ==I;
      );
      =     #INTERNAL.IF.Silo.SiloNr_correct;
      A     #HMI.CMD.StartFeeding;
      AN    #INTERNAL.IF.Silo.SiloNr_correct;
      FP    #INTERNAL.Flags.FP_Start_wo_Silocorrect.helpBit;
      =     #INTERNAL.Flags.FP_Start_wo_Silocorrect.pulseBit;
      A     #INTERNAL.Flags.FP_Start_wo_Silocorrect.pulseBit;
      S     #fSiloNrNotCorrect;
      A     #INTERNAL.IF.Silo.SiloNr_correct;
      O     #aSiloNrNotCorrect;	// ak
      R     #fSiloNrNotCorrect;
NETWORK
TITLE = Filling: Change Silo Nr not possible-blocking
      A(;
      L     #HMI.PARAM.StorageLocation;
      L     #HMI.PV.StorageLocation;
      <>I;
      );
      A(;
      ON    #INTERNAL.Flags.StatusHP03.HP03_empty;
      ON    #INTERNAL.Flags.StatusREC01.REC01_empty;
      O     #INTERNAL.Flags.ReleaseFeeding;
      );
      S     #HMI.STATE.ChangingHpBlocked;
      A     #INTERNAL.Flags.StatusHP03.HP03_empty;
      A     #INTERNAL.Flags.StatusREC01.REC01_empty;
      AN    #INTERNAL.Flags.ReleaseFeeding;
      O;
      A(;
      L     #HMI.PARAM.StorageLocation;
      L     #HMI.PV.StorageLocation;
      ==I;
      );
      R     #HMI.STATE.ChangingHpBlocked;
      A     #HMI.STATE.ChangingHpBlocked;
      A(;
      L     #HMI.PARAM.StorageLocation;
      L     0;
      <>I;
      );
      =     #fLineNotEmpty;
NETWORK
TITLE = Filling: Filling RELEASE set/reset
      A     #SEQUENCE.Filling.AUTO;
      A     #INTERNAL.Flags.ReleaseFeeding;
      A     #INTERNAL.IF.Silo.SiloNr_correct;
      AN    #LevelIndicators.HighLevelREC01.debounced_covered;
      FP    #INTERNAL.Flags.FP_releaseFilling.helpBit;
      =     #INTERNAL.Flags.FP_releaseFilling.pulseBit;
      A     #INTERNAL.Flags.FP_releaseFilling.pulseBit;
      S     #SEQUENCE.Filling.RELEASE;
      AN    #INTERNAL.Flags.ReleaseFeeding;
      A     #INTERNAL.Flags.CleaningFinished;
      AN    #LevelIndicators.HighLevelREC01.debounced_covered;
      AN    #LevelIndicators.HighLevelHP03.debounced_covered;
//      ON    #iSystemActive
      R     #SEQUENCE.Filling.RELEASE;
NETWORK
TITLE = Filling: request blower
      O     #SEQUENCE.Filling.RELEASE;
      O     #INTERNAL.Flags.CleaningRelease;
      =     #IF_Blower.CONTROL.CMD.Request;
NETWORK
TITLE = Filling: request storage location
      A     #SEQUENCE.Filling.RELEASE;
      A     #IF_Blower.STATUS.STATE.Active;
      =     #IF_Silo.CONTROL.CMD.Request;
NETWORK
TITLE = Filling: release blower
      A(;
      A     #SEQUENCE.Filling.RELEASE;
      AN    #fREC01HighLevel;
      O;
      A     #INTERNAL.Flags.CleaningRelease;
      );
      A     #IF_Blower.STATUS.STATE.Ready;
      =     #IF_Blower.CONTROL.CMD.Release;
NETWORK
TITLE = Filling: release storage location
      A     #SEQUENCE.Filling.RELEASE;
      AN    #INTERNAL.Flags.CleaningRelease;
      A     #IF_Silo.STATUS.STATE.Ready;
      A     #IF_Blower.STATUS.STATE.Active;
//     A     #INTERNAL.Flags.PressureBuilt
      AN    #LevelIndicators.HighLevelREC01.debounced_covered;
      AN    #LevelIndicators.HighLevelHP03.debounced_covered;
      AN    #IF_Blower.STATUS.STATE.PressureFault;
      AN    #INTERNAL.Flags.StatusREC01.REC01_LowLevelCovered;
      AN    #fREC01HighLevel;
      A     #INTERNAL.Flags.StatusHP03.HP03_HL_disclosured;	// ak
      =     #IF_Silo.CONTROL.CMD.Release;
NETWORK
TITLE = Filling: release filter
      A     #SEQUENCE.Filling.ACTIVE;
      A     #IF_Blower.STATUS.STATE.Active;	// ak
      A     #IF_Silo.STATUS.STATE.Active;	// ak
      =     #PurgedFilter.auto_mode_control_clock1;
      O     #SEQUENCE.Filling.AUTO;
      O     #SEQUENCE.Discharging.AUTO;
      A(;
      O     #SEQUENCE.Discharging.ACTIVE;
      O     #SEQUENCE.Filling.ACTIVE;
      );
      AN    "Service mode lock auto";
      =     #PurgedFilter.man_mode_locked;
NETWORK
TITLE = Filling: FILLING ACTIVE
      A     #SEQUENCE.Filling.RELEASE;
      A     #IF_Blower.STATUS.STATE.Active;
      A     #IF_Silo.STATUS.STATE.Active;
      =     #SEQUENCE.Filling.ACTIVE;
NETWORK
TITLE = -----------------Cleaning-------------------
NETWORK
TITLE = Cleaning: Cleaning release and finish
      A     #iSystemActive;
      A     #SEQUENCE.Filling.AUTO;
      A(;
      AN    #HMI.CMD.StartFeeding;
      A     #IF_Blower.STATUS.STATE.EmptyPressure;
      AN    #INTERNAL.Flags.StatusREC01.REC01_empty;
      O;
      A     #HMI.CMD.StartFeeding;
      A     #LevelIndicators.HighLevelREC01.debounced_covered;
      );
      FP    #INTERNAL.Flags.FP_CleaningRelease.helpBit;
      S     #INTERNAL.Flags.CleaningRelease;
      A     #INTERNAL.Flags.CleaningRelease;
      =     #HMI.STATE.cleaning_active;
      A     #INTERNAL.Flags.CleaningRelease;
      =     #TIMERS.TV_CleaningLineDuration.IN;
      ON    #iSystemActive;
      =     #TIMERS.TV_CleaningLineDuration.RST;
      CALL  "FC3 Cycle generator" (
           in_Freigabe              := #TIMERS.TV_CleaningLineDuration.IN,
           in_Reset                 := #TIMERS.TV_CleaningLineDuration.RST,
           in_Impuls                := "M 1.7 Cycle Timer-FC",
           in_Impulszeit_in_100ms   := "MW 6 Timer Val Cycle FCs",
           in_Verzoegerungsart      := B#16#56,
           in_Verzoegerungszeit     := #HMI.PARAM.CleaningDuration,
           io_Ausgangssignal        := #TIMERS.TV_CleaningLineDuration.Q,
           io_Zeitzaehler           := #TIMERS.TV_CleaningLineDuration.ET);
      L     #TIMERS.TV_CleaningLineDuration.ET;
      T     #HMI.PV.CleaningDuration;
      A     #INTERNAL.Flags.CleaningRelease;
//     A     #IF_Blower.STATUS.STATE.EmptyPressure
      AN    #TIMERS.TV_CleaningLineDuration.Q;
      R     #INTERNAL.Flags.CleaningRelease;
      AN    #INTERNAL.Flags.CleaningRelease;
      A(;
      A     #HMI.CMD.StartFeeding;
      AN    #fREC01HighLevel;
      O;
      AN    #HMI.CMD.StartFeeding;
      );
      =     #INTERNAL.Flags.CleaningFinished;
NETWORK
TITLE = --------------------- Sequence Discharging ---------------------
NETWORK
TITLE = Discharging: discharging is forbidden from VISU
      A     #HMI.CMD.REC01_disch_forbidden;
      =     #INTERNAL.Flags.DischargeREC01_forbidden;
NETWORK
TITLE = Discharging: Filling HP03 is blocked with delay variable
      A     #LevelIndicators.HighLevelHP03.debounced_covered;
      S     #INTERNAL.Flags.StatusHP03.filling_locked;
      AN    #LevelIndicators.HighLevelHP03.debounced_covered;
      AN    #LevelIndicators.LowLevelHP03.debounced_covered;
      O;
      AN    #LevelIndicators.HighLevelHP03.debounced_covered;
      A     #TIMERS.TON_HP03_HL_DISCLOSURE.Q;
      R     #INTERNAL.Flags.StatusHP03.filling_locked;
NETWORK
TITLE = Discharging: Disclosure of High Level HP03
      A     #LevelIndicators.HighLevelHP03.debounced_covered;	// ak
      R     #INTERNAL.Flags.StatusHP03.HP03_HL_disclosured;	// ak
      A     #INTERNAL.Flags.StatusHP03.filling_locked;
      AN    #LevelIndicators.HighLevelHP03.debounced_covered;
      A     #iPFCPM_TakeProduct;
      =     #TIMERS.TON_HP03_HL_DISCLOSURE.IN;
      AN    #iSystemActive;
      =     #TIMERS.TON_HP03_HL_DISCLOSURE.RST;
      CALL  "FC3 Cycle generator" (
           in_Freigabe              := #TIMERS.TON_HP03_HL_DISCLOSURE.IN,
           in_Reset                 := #TIMERS.TON_HP03_HL_DISCLOSURE.RST,
           in_Impuls                := "M 1.7 Cycle Timer-FC",
           in_Impulszeit_in_100ms   := "MW 6 Timer Val Cycle FCs",
           in_Verzoegerungsart      := B#16#45,
           in_Verzoegerungszeit     := #HMI.PARAM.DelayHighLevelHP03,
           io_Ausgangssignal        := #TIMERS.TON_HP03_HL_DISCLOSURE.Q,
           io_Zeitzaehler           := #TIMERS.TON_HP03_HL_DISCLOSURE.ET);
      A     #TIMERS.TON_HP03_HL_DISCLOSURE.Q;
      O;
      AN    #LevelIndicators.HighLevelHP03.debounced_covered;	// ak
      AN    #LevelIndicators.LowLevelHP03.debounced_covered;	// ak
      S     #INTERNAL.Flags.StatusHP03.HP03_HL_disclosured;	// ak
      L     #TIMERS.TON_HP03_HL_DISCLOSURE.ET;
      T     #HMI.PV.DelayHP03HighLevel;
NETWORK
TITLE = Discharging: discharging RELEASE
      A     #SEQUENCE.Discharging.AUTO;
      A     #iSystemActive;
      AN    #LevelIndicators.HighLevelHP03.debounced_covered;
      AN    #fRepRotaryValve;
      AN    #fRepScreener;
      AN    #fRepMetalSeparator;
      AN    #fRepMetalSeparator;
      AN    #fSafetyRotaryFeeder;
      AN    #fSafetyMS;
      AN    #HMI.CMD.REC01_disch_forbidden;	// from VISU only for test
      AN    #INTERNAL.Flags.DischargeREC01_forbidden;
      A(;
      O     #INTERNAL.Flags.ReleaseFeeding;
      O     #INTERNAL.Flags.StatusREC01.REC01_material_signal;
      );
      =     #SEQUENCE.Discharging.RELEASE;
NETWORK
TITLE = Discharging: release metal separator
      A     #SEQUENCE.Discharging.AUTO;
      A     #SEQUENCE.Discharging.RELEASE;
      AN    #INTERNAL.Flags.DischargeREC01_forbidden;
      A(;
      A     #INTERNAL.Flags.StatusHP03.HP03_HL_disclosured;
      O;
      AN    #LevelIndicators.HighLevelHP03.debounced_covered;
      AN    #LevelIndicators.LowLevelHP03.debounced_covered;
      );
      =     #TIMERS.TOF_MetalSeparator_Delay.IN;
// delay off metal separator motor
      ON    #iRepMetalSeparator_on;
      ON    #iSystemActive;
      =     #TIMERS.TOF_MetalSeparator_Delay.RST;
      CALL  "FC3 Cycle generator" (
           in_Freigabe              := #TIMERS.TOF_MetalSeparator_Delay.IN,
           in_Reset                 := #TIMERS.TOF_MetalSeparator_Delay.RST,
           in_Impuls                := "M 1.7 Cycle Timer-FC",
           in_Impulszeit_in_100ms   := "MW 6 Timer Val Cycle FCs",
           in_Verzoegerungsart      := B#16#41,
           in_Verzoegerungszeit     := #HMI.PARAM.DelayScreener,
           io_Ausgangssignal        := #TIMERS.TOF_MetalSeparator_Delay.Q,
           io_Zeitzaehler           := #TIMERS.TOF_MetalSeparator_Delay.ET);
      A     #TIMERS.TOF_MetalSeparator_Delay.Q;
      =     #MetalSeparator.auto_mode_control;
      L     #TIMERS.TOF_MetalSeparator_Delay.ET;
      T     #HMI.PV.DelayScreener;
NETWORK
TITLE = Discharging: Metal separator object
      A     #SEQUENCE.Discharging.AUTO;
      AN    "Service mode lock auto";
      A     #SEQUENCE.Discharging.ACTIVE;
      =     #MetalSeparator.man_mode_locked;
      O     #fSafetyMS;
      O     #fRepMetalSeparator;
      =     #MetalSeparator.motor_locked;
      CALL  "FC20 Motor 1O1I" (
           in_Handbedienung_erlaubt := TRUE,
           in_Quitt_Stoerung_noetig := TRUE,
           in_Anlage_ein            := #iSystemActive,
           in_Quitt_Stoerung        := #aFBMetalSeparator,
           in_Ansteuerung_Motor     := #MetalSeparator.auto_mode_control,
           in_Eingang_Motor         := #iFBMetalSeparator_on,
           io_Ausgang_Motor         := #qMetalSeparator_on,
           io_Motor_in_Betrieb      := #MetalSeparator.motor_in_operation,
           io_Stoerung              := #fFBMetalSeparator,
           io_Motorstruktur         := #MetalSeparator);
NETWORK
TITLE = Discharging: release screener
      A     #SEQUENCE.Discharging.AUTO;
      A     #SEQUENCE.Discharging.RELEASE;
      A     #MetalSeparator.motor_in_operation;
      AN    #HMI.CMD.REC01_disch_forbidden;
      AN    #LevelIndicators.HighLevelHP03.debounced_covered;
      =     #TIMERS.TOF_Screener_Delay.IN;
      ON    #iRepScreener_on;
      ON    #iSystemActive;
      =     #TIMERS.TOF_Screener_Delay.RST;
      CALL  "FC3 Cycle generator" (
           in_Freigabe              := #TIMERS.TOF_Screener_Delay.IN,
           in_Reset                 := #TIMERS.TOF_Screener_Delay.RST,
           in_Impuls                := "M 1.7 Cycle Timer-FC",
           in_Impulszeit_in_100ms   := "MW 6 Timer Val Cycle FCs",
           in_Verzoegerungsart      := B#16#41,
           in_Verzoegerungszeit     := #HMI.PARAM.DelayScreener,
           io_Ausgangssignal        := #TIMERS.TOF_Screener_Delay.Q,
           io_Zeitzaehler           := #TIMERS.TOF_Screener_Delay.ET);
      A     #TIMERS.TOF_Screener_Delay.Q;
      =     #Screener.auto_mode_control;
NETWORK
TITLE = Discharging: Screener object
      A     #SEQUENCE.Discharging.AUTO;
      AN    "Service mode lock auto";
      A     #SEQUENCE.Discharging.ACTIVE;
      =     #Screener.man_mode_locked;
      O     #fRepScreener;
      =     #Screener.motor_locked;
      CALL  "FC20 Motor 1O1I" (
           in_Handbedienung_erlaubt := TRUE,
           in_Quitt_Stoerung_noetig := TRUE,
           in_Anlage_ein            := #iSystemActive,
           in_Quitt_Stoerung        := #aFBScreener,
           in_Ansteuerung_Motor     := #Screener.auto_mode_control,
           in_Eingang_Motor         := #iFBScreener_on,
           io_Ausgang_Motor         := #qScreener_on,
           io_Motor_in_Betrieb      := #Screener.motor_in_operation,
           io_Stoerung              := #fFBScreener,
           io_Motorstruktur         := #Screener);
NETWORK
TITLE = Discharging: release air purged bearing rotary valve
      A     #SEQUENCE.Discharging.AUTO;
      A     #SEQUENCE.Discharging.RELEASE;
      AN    #HMI.CMD.REC01_disch_forbidden;	// ak
      AN    #LevelIndicators.HighLevelHP03.debounced_covered;
      A     #Screener.motor_in_operation;
      A     #MetalSeparator.motor_in_operation;
      AN    #fToolKeyControl;
      AN    #fSafetyRotaryFeeder;
      =     #TIMERS.TOF_AirPurgedBearing.IN;
      O     #fSafetyRotaryFeeder;
      ON    #iSystemActive;
      =     #TIMERS.TOF_AirPurgedBearing.RST;
      CALL  "FC3 Cycle generator" (
           in_Freigabe              := #TIMERS.TOF_AirPurgedBearing.IN,
           in_Reset                 := #TIMERS.TOF_AirPurgedBearing.RST,
           in_Impuls                := "M 1.7 Cycle Timer-FC",
           in_Impulszeit_in_100ms   := "MW 6 Timer Val Cycle FCs",
           in_Verzoegerungsart      := B#16#41,
           in_Verzoegerungszeit     := 1.500000e+00,
           io_Ausgangssignal        := #TIMERS.TOF_AirPurgedBearing.Q,
           io_Zeitzaehler           := #TIMERS.TOF_AirPurgedBearing.ET);	// 1.000000e+000 ak
      A     #TIMERS.TOF_AirPurgedBearing.Q;
      =     #AirPurgedBearing.auto_mode_control;
NETWORK
TITLE = Discharging: Air purge bearing object
      A     #SEQUENCE.Discharging.AUTO;
      AN    "Service mode lock auto";
      A     #SEQUENCE.Discharging.ACTIVE;
      =     #AirPurgedBearing.man_mode_locked;
      CALL  "FC21 Valve 10-2I" (
           in_Ventil_Typ            := 0,
           in_Handbedienung_erlaubt := TRUE,
           in_Quitt_Stoerung_noetig := FALSE,
           in_Quitt_Stoerung        := FALSE,
           in_Anlage_ein            := #iSystemActive,
           in_Ansteuerung_Ventil    := #AirPurgedBearing.auto_mode_control,
           in_Eingang_angesteuert   := #AirPurgedBearing.input_valve_set,
           in_Eingang_nicht_angest  := #AirPurgedBearing.input_valve_not_set,
           io_Ausgang_Ventil        := #qAPBRotaryValve_on,
           io_Ventil_in_Betrieb     := #AirPurgedBearing.valve_in_operation,
           io_Stoerung              := #AirPurgedBearing.fault,
           io_Ventilstruktur        := #AirPurgedBearing);
NETWORK
TITLE = Discharging: release rotary feeder
      A     #SEQUENCE.Discharging.AUTO;
      A     #SEQUENCE.Discharging.RELEASE;
      AN    #HMI.CMD.REC01_disch_forbidden;	// ak
      AN    #LevelIndicators.HighLevelHP03.debounced_covered;
      A     #Screener.motor_in_operation;
      A     #MetalSeparator.motor_in_operation;
      A     #AirPurgedBearing.valve_in_operation;
      =     #RotaryFeeder.auto_mode_control;
NETWORK
TITLE = Discharging: Rotary Valve object
      A     #SEQUENCE.Discharging.AUTO;
      AN    "Service mode lock auto";
      A     #SEQUENCE.Discharging.ACTIVE;
      =     #RotaryFeeder.man_mode_locked;
      O     #fSafetyRotaryFeeder;
      O     #fToolKeyControl;
      O     #fRepRotaryValve;
      =     #RotaryFeeder.motor_locked;
      CALL  "FC20 Motor 1O1I" (
           in_Handbedienung_erlaubt := TRUE,
           in_Quitt_Stoerung_noetig := TRUE,
